C01781=1037.136,384.504,-134.094,173.331,45.031,158.902
C01782=1037.127,384.258,-134.052,173.323,45.027,158.900
C01783=1037.118,384.011,-134.010,173.315,45.023,158.898
C01784=1037.109,383.766,-133.968,173.307,45.019,158.896
C01785=1037.100,383.519,-133.926,173.300,45.015,158.895
C01786=1037.091,383.273,-133.884,173.291,45.011,158.893
C01787=1037.082,383.027,-133.842,173.284,45.007,158.891
C01788=1037.075,382.781,-133.800,173.277,45.004,158.889
C01789=1037.066,382.534,-133.759,173.268,45.000,158.888
C01790=1037.057,382.288,-133.717,173.261,44.996,158.886
C01791=1037.048,382.042,-133.675,173.253,44.991,158.884
C01792=1037.039,381.795,-133.634,173.245,44.988,158.882
C01793=1037.031,381.549,-133.593,173.238,44.984,158.881
C01794=1037.022,381.303,-133.551,173.230,44.980,158.879
C01795=1037.014,381.056,-133.509,173.222,44.976,158.877
C01796=1037.006,380.810,-133.468,173.215,44.972,158.875
C01797=1036.997,380.564,-133.426,173.208,44.968,158.874
C01798=1036.988,380.317,-133.385,173.199,44.965,158.872
C01799=1036.979,380.070,-133.343,173.192,44.961,158.870
C01800=1036.971,379.825,-133.302,173.185,44.957,158.869
C01801=1036.962,379.578,-133.261,173.177,44.953,158.867
C01802=1036.954,379.332,-133.219,173.169,44.950,158.865
C01803=1036.946,379.085,-133.177,173.162,44.946,158.863
C01804=1036.937,378.839,-133.136,173.155,44.942,158.862
C01805=1036.923,378.436,-133.069,173.142,44.936,158.859
C01806=1036.909,378.034,-133.001,173.131,44.930,158.856
C01807=1036.895,377.630,-132.935,173.118,44.924,158.854
C01808=1036.881,377.228,-132.867,173.107,44.918,158.851
C01809=1036.872,376.982,-132.827,173.099,44.915,158.849
C01810=1036.864,376.735,-132.786,173.091,44.911,158.848
C01811=1036.855,376.488,-132.745,173.084,44.907,158.846
C01812=1036.847,376.242,-132.705,173.077,44.904,158.844
C01813=1036.838,375.996,-132.663,173.070,44.900,158.843
C01814=1036.829,375.750,-132.623,173.063,44.896,158.841
C01815=1036.821,375.503,-132.582,173.055,44.893,158.839
C01816=1036.813,375.256,-132.541,173.047,44.889,158.838
C01817=1036.805,375.010,-132.501,173.040,44.886,158.836
C01818=1036.796,374.763,-132.460,173.033,44.883,158.835
C01819=1036.787,374.517,-132.420,173.026,44.879,158.833
C01820=1036.779,374.270,-132.379,173.019,44.876,158.832
C01821=1036.771,374.024,-132.338,173.012,44.872,158.830
C01822=1036.763,373.778,-132.297,173.005,44.869,158.828
C01823=1036.753,373.531,-132.257,172.998,44.865,158.827
C01824=1036.746,373.284,-132.217,172.991,44.862,158.825
C01825=1036.738,373.038,-132.176,172.984,44.858,158.824
C01826=1036.729,372.791,-132.135,172.976,44.855,158.822
C01827=1036.721,372.545,-132.095,172.969,44.851,158.821
C01828=1036.712,372.298,-132.056,172.962,44.848,158.819
C01829=1036.704,372.052,-132.015,172.955,44.845,158.818
C01830=1036.696,371.805,-131.974,172.948,44.841,158.816
C01831=1036.688,371.558,-131.933,172.941,44.838,158.815
C01832=1036.679,371.312,-131.894,172.934,44.835,158.813
C01833=1036.671,371.066,-131.853,172.927,44.832,158.812
C01834=1036.664,370.819,-131.813,172.921,44.828,158.810
C01835=1036.655,370.572,-131.772,172.914,44.825,158.809
C01836=1036.647,370.325,-131.733,172.907,44.821,158.807
C01837=1036.639,370.079,-131.692,172.900,44.818,158.806
C01838=1036.631,369.832,-131.652,172.893,44.814,158.804
C01839=1036.622,369.586,-131.612,172.886,44.811,158.803
C01840=1036.614,369.339,-131.573,172.879,44.808,158.801
C01841=1036.605,369.092,-131.533,172.872,44.805,158.800
C01842=1036.596,368.846,-131.493,172.865,44.802,158.798
C01843=1036.589,368.599,-131.453,172.859,44.799,158.797
C01844=1036.580,368.352,-131.414,172.852,44.796,158.795
C01845=1036.573,368.105,-131.374,172.845,44.792,158.794
C01846=1036.564,367.859,-131.334,172.838,44.789,158.792
C01847=1036.556,367.612,-131.294,172.831,44.786,158.791
C01848=1036.548,367.366,-131.254,172.825,44.783,158.790
C01849=1036.539,367.119,-131.215,172.818,44.780,158.788
C01850=1036.531,366.872,-131.175,172.811,44.777,158.787
C01851=1036.523,366.626,-131.136,172.805,44.774,158.785
C01852=1036.515,366.379,-131.096,172.798,44.771,158.784
C01853=1036.507,366.132,-131.057,172.791,44.768,158.782
C01854=1036.499,365.885,-131.017,172.785,44.764,158.781
C01855=1036.491,365.639,-130.977,172.778,44.761,158.780
C01856=1036.482,365.392,-130.938,172.771,44.758,158.778
C01857=1036.474,365.145,-130.898,172.765,44.755,158.777
C01858=1036.466,364.899,-130.859,172.758,44.752,158.775
C01859=1036.459,364.651,-130.820,172.752,44.749,158.774
C01860=1036.450,364.404,-130.780,172.745,44.746,158.773
C01861=1036.438,364.022,-130.719,172.734,44.741,158.770
C01862=1036.426,363.640,-130.658,172.725,44.737,158.768
C01863=1036.413,363.258,-130.598,172.715,44.732,158.766
C01864=1036.401,362.876,-130.537,172.704,44.728,158.764
C01865=1036.393,362.629,-130.497,172.698,44.724,158.763
C01866=1036.385,362.382,-130.458,172.692,44.721,158.761
C01867=1036.377,362.136,-130.419,172.685,44.719,158.760
C01868=1036.369,361.889,-130.379,172.679,44.716,158.759
C01869=1036.361,361.642,-130.341,172.672,44.712,158.757
C01870=1036.353,361.395,-130.301,172.666,44.710,158.756
C01871=1036.345,361.148,-130.263,172.659,44.707,158.755
C01872=1036.338,360.901,-130.224,172.653,44.704,158.754
C01873=1036.329,360.654,-130.185,172.647,44.701,158.752
C01874=1036.321,360.407,-130.146,172.640,44.699,158.751
C01875=1036.313,360.161,-130.107,172.634,44.695,158.750
C01876=1036.305,359.914,-130.069,172.628,44.693,158.748
C01877=1036.297,359.667,-130.030,172.621,44.691,158.747
C01878=1036.289,359.420,-129.992,172.615,44.687,158.746
C01879=1036.281,359.174,-129.952,172.609,44.685,158.745
C01880=1036.274,358.926,-129.913,172.603,44.681,158.743
C01881=1036.266,358.680,-129.875,172.596,44.679,158.742
C01882=1036.258,358.432,-129.836,172.590,44.676,158.741
C01883=1036.250,358.185,-129.798,172.584,44.674,158.740
C01884=1036.242,357.939,-129.759,172.577,44.671,158.738
C01885=1036.234,357.691,-129.721,172.571,44.668,158.737
C01886=1036.226,357.446,-129.682,172.565,44.666,158.736
C01887=1036.218,357.198,-129.643,172.559,44.663,158.734
C01888=1036.210,356.952,-129.605,172.553,44.660,158.733
C01889=1036.202,356.705,-129.566,172.546,44.657,158.732
C01890=1036.195,356.458,-129.528,172.541,44.655,158.731
C01891=1036.187,356.211,-129.490,172.534,44.652,158.729
C01892=1036.179,355.964,-129.452,172.529,44.649,158.728
C01893=1036.171,355.717,-129.413,172.522,44.647,158.727
C01894=1036.163,355.469,-129.375,172.516,44.644,158.726
C01895=1036.155,355.223,-129.337,172.510,44.642,158.725
C01896=1036.147,354.976,-129.298,172.504,44.639,158.723
C01897=1036.140,354.728,-129.260,172.498,44.636,158.722
C01898=1036.132,354.482,-129.223,172.491,44.634,158.721
C01899=1036.124,354.235,-129.184,172.486,44.631,158.720
C01900=1036.116,353.989,-129.146,172.479,44.629,158.719
C01901=1036.108,353.741,-129.108,172.474,44.626,158.717
C01902=1036.101,353.494,-129.070,172.467,44.624,158.716
C01903=1036.093,353.246,-129.032,172.462,44.621,158.715
C01904=1036.085,353.000,-128.994,172.455,44.618,158.714
C01905=1036.077,352.754,-128.956,172.450,44.616,158.713
C01906=1036.069,352.506,-128.918,172.443,44.614,158.711
C01907=1036.062,352.259,-128.880,172.438,44.611,158.710
C01908=1036.054,352.012,-128.842,172.432,44.608,158.709
C01909=1036.046,351.765,-128.804,172.426,44.606,158.708
C01910=1036.039,351.518,-128.766,172.420,44.604,158.707
C01911=1036.031,351.271,-128.728,172.414,44.601,158.706
C01912=1036.023,351.024,-128.691,172.408,44.598,158.704
C01913=1036.015,350.777,-128.652,172.402,44.596,158.703
C01914=1036.008,350.530,-128.615,172.396,44.594,158.702
C01915=1036.001,350.283,-128.577,172.391,44.591,158.701
C01916=1035.993,350.036,-128.539,172.385,44.589,158.700
C01917=1035.981,349.660,-128.482,172.376,44.585,158.698
C01918=1035.969,349.284,-128.425,172.367,44.581,158.696
C01919=1035.957,348.907,-128.368,172.358,44.578,158.695
C01920=1035.946,348.531,-128.311,172.350,44.574,158.693
C01921=1035.938,348.284,-128.273,172.343,44.572,158.692
C01922=1035.931,348.037,-128.235,172.338,44.570,158.691
C01923=1035.923,347.790,-128.198,172.333,44.567,158.690
C01924=1035.916,347.543,-128.161,172.326,44.565,158.689
C01925=1035.908,347.296,-128.124,172.321,44.563,158.688
C01926=1035.900,347.048,-128.086,172.315,44.560,158.686
C01927=1035.893,346.801,-128.048,172.309,44.558,158.685
C01928=1035.885,346.554,-128.011,172.304,44.556,158.684
C01929=1035.877,346.307,-127.974,172.298,44.553,158.683
C01930=1035.869,346.060,-127.937,172.292,44.551,158.682
C01931=1035.862,345.813,-127.899,172.287,44.549,158.681
C01932=1035.854,345.566,-127.863,172.281,44.547,158.680
C01933=1035.847,345.319,-127.826,172.275,44.545,158.679
C01934=1035.840,345.072,-127.788,172.270,44.542,158.678
C01935=1035.832,344.825,-127.751,172.264,44.540,158.677
C01936=1035.825,344.578,-127.714,172.259,44.538,158.676
C01937=1035.817,344.330,-127.677,172.253,44.536,158.675
C01938=1035.810,344.083,-127.640,172.247,44.533,158.674
C01939=1035.802,343.836,-127.603,172.242,44.531,158.673
C01940=1035.795,343.589,-127.566,172.237,44.529,158.672
C01941=1035.787,343.342,-127.529,172.230,44.527,158.671
C01942=1035.780,343.094,-127.492,172.225,44.525,158.670
C01943=1035.772,342.848,-127.455,172.220,44.522,158.668
C01944=1035.764,342.600,-127.419,172.214,44.520,158.667
C01945=1035.757,342.353,-127.381,172.208,44.518,158.666
C01946=1035.749,342.106,-127.345,172.203,44.516,158.665
C01947=1035.742,341.858,-127.307,172.197,44.514,158.664
C01948=1035.734,341.611,-127.271,172.192,44.512,158.663
C01949=1035.727,341.364,-127.234,172.187,44.510,158.662
C01950=1035.719,341.116,-127.197,172.181,44.508,158.661
C01951=1035.712,340.870,-127.161,172.175,44.506,158.660
C01952=1035.705,340.623,-127.124,172.170,44.503,158.659
C01953=1035.697,340.376,-127.087,172.165,44.502,158.658
C01954=1035.689,340.128,-127.051,172.160,44.500,158.657
C01955=1035.682,339.881,-127.015,172.153,44.498,158.656
C01956=1035.674,339.634,-126.977,172.148,44.496,158.655
C01957=1035.667,339.386,-126.941,172.143,44.493,158.654
C01958=1035.660,339.140,-126.905,172.138,44.492,158.653
C01959=1035.652,338.892,-126.869,172.133,44.490,158.652
C01960=1035.644,338.645,-126.832,172.127,44.488,158.651
C01961=1035.637,338.397,-126.795,172.121,44.486,158.650
C01962=1035.629,338.150,-126.759,172.116,44.483,158.649
C01963=1035.622,337.903,-126.723,172.111,44.482,158.649
C01964=1035.615,337.656,-126.687,172.106,44.480,158.647
C01965=1035.608,337.408,-126.650,172.100,44.477,158.646
C01966=1035.600,337.161,-126.614,172.095,44.476,158.646
C01967=1035.593,336.915,-126.577,172.090,44.474,158.645
C01968=1035.585,336.667,-126.541,172.085,44.472,158.644
C01969=1035.577,336.420,-126.505,172.080,44.470,158.643
C01970=1035.570,336.172,-126.468,172.073,44.468,158.642
C01971=1035.563,335.925,-126.432,172.068,44.466,158.641
C01972=1035.556,335.678,-126.396,172.063,44.464,158.640
C01973=1035.545,335.298,-126.340,172.055,44.461,158.638
C01974=1035.533,334.919,-126.285,172.048,44.458,158.637
C01975=1035.522,334.538,-126.230,172.040,44.455,158.636
C01976=1035.511,334.159,-126.175,172.031,44.453,158.634
C01977=1035.503,333.911,-126.138,172.026,44.451,158.633
C01978=1035.496,333.665,-126.103,172.021,44.449,158.632
C01979=1035.489,333.417,-126.067,172.016,44.447,158.631
C01980=1035.481,333.170,-126.031,172.010,44.445,158.630
C01981=1035.474,332.922,-125.995,172.005,44.444,158.630
C01982=1035.466,332.675,-125.959,172.000,44.442,158.629
C01983=1035.459,332.428,-125.924,171.995,44.440,158.628
C01984=1035.451,332.180,-125.888,171.990,44.438,158.627
C01985=1035.444,331.934,-125.852,171.985,44.437,158.626
C01986=1035.437,331.686,-125.817,171.980,44.435,158.625
C01987=1035.429,331.439,-125.781,171.975,44.433,158.624
C01988=1035.422,331.191,-125.745,171.970,44.431,158.623
C01989=1035.415,330.944,-125.710,171.964,44.429,158.622
C01990=1035.408,330.696,-125.674,171.959,44.428,158.622
C01991=1035.401,330.449,-125.638,171.954,44.426,158.621
C01992=1035.393,330.202,-125.602,171.949,44.424,158.620
C01993=1035.386,329.955,-125.567,171.944,44.423,158.619
C01994=1035.379,329.706,-125.531,171.939,44.421,158.618
C01995=1035.372,329.460,-125.495,171.934,44.419,158.617
C01996=1035.364,329.212,-125.460,171.929,44.418,158.616
C01997=1035.357,328.965,-125.424,171.924,44.416,158.616
C01998=1035.350,328.718,-125.389,171.919,44.414,158.615
C01999=1035.342,328.470,-125.353,171.914,44.412,158.614
C02000=1035.335,328.223,-125.318,171.909,44.411,158.613
C02001=1035.328,327.975,-125.283,171.904,44.409,158.612
C02002=1035.320,327.728,-125.248,171.899,44.407,158.611
C02003=1035.313,327.480,-125.213,171.894,44.406,158.610
C02004=1035.305,327.233,-125.177,171.890,44.404,158.610
C02005=1035.298,326.986,-125.142,171.885,44.403,158.609
C02006=1035.290,326.738,-125.107,171.880,44.401,158.608
C02007=1035.284,326.491,-125.072,171.875,44.400,158.607
C02008=1035.275,326.243,-125.037,171.870,44.398,158.606
C02009=1035.269,325.996,-125.002,171.865,44.397,158.606
C02010=1035.261,325.749,-124.968,171.860,44.395,158.605
C02011=1035.254,325.501,-124.932,171.855,44.394,158.604
C02012=1035.246,325.254,-124.898,171.850,44.392,158.603
C02013=1035.240,325.006,-124.862,171.845,44.390,158.602
C02014=1035.231,324.758,-124.828,171.840,44.389,158.602
C02015=1035.225,324.511,-124.792,171.835,44.388,158.601
C02016=1035.217,324.264,-124.758,171.830,44.386,158.600
C02017=1035.210,324.016,-124.722,171.826,44.384,158.599
C02018=1035.202,323.769,-124.688,171.821,44.383,158.598
C02019=1035.196,323.522,-124.653,171.816,44.382,158.598
C02020=1035.188,323.275,-124.618,171.811,44.380,158.597
C02021=1035.181,323.026,-124.583,171.806,44.379,158.596
C02022=1035.173,322.779,-124.548,171.801,44.377,158.595
C02023=1035.167,322.531,-124.514,171.796,44.376,158.594
C02024=1035.159,322.284,-124.479,171.791,44.374,158.594
C02025=1035.152,322.036,-124.444,171.787,44.373,158.593
C02026=1035.144,321.789,-124.409,171.783,44.372,158.592
C02027=1035.138,321.542,-124.374,171.778,44.370,158.591
C02028=1035.130,321.294,-124.340,171.773,44.368,158.590
C02029=1035.119,320.910,-124.286,171.765,44.366,158.589
C02030=1035.108,320.526,-124.232,171.758,44.364,158.588
C02031=1035.096,320.142,-124.178,171.750,44.362,158.587
C02032=1035.085,319.757,-124.125,171.743,44.360,158.586
C02033=1035.079,319.510,-124.090,171.739,44.358,158.585
C02034=1035.071,319.262,-124.056,171.734,44.357,158.584
C02035=1035.065,319.015,-124.021,171.729,44.356,158.584
C02036=1035.057,318.767,-123.987,171.724,44.354,158.583
C02037=1035.051,318.519,-123.952,171.720,44.353,158.582
C02038=1035.043,318.272,-123.918,171.715,44.351,158.581
C02039=1035.037,318.024,-123.883,171.711,44.350,158.581
C02040=1035.029,317.777,-123.849,171.706,44.349,158.580
C02041=1035.022,317.530,-123.814,171.701,44.347,158.579
C02042=1035.015,317.282,-123.780,171.697,44.346,158.578
C02043=1035.008,317.035,-123.746,171.692,44.344,158.577
C02044=1035.001,316.787,-123.711,171.687,44.343,158.577
C02045=1034.994,316.540,-123.677,171.683,44.342,158.576
C02046=1034.987,316.292,-123.642,171.678,44.340,158.575
C02047=1034.980,316.045,-123.608,171.673,44.339,158.575
C02048=1034.973,315.798,-123.573,171.668,44.338,158.574
C02049=1034.966,315.550,-123.539,171.665,44.337,158.573
C02050=1034.959,315.302,-123.505,171.660,44.335,158.572
C02051=1034.952,315.055,-123.470,171.655,44.334,158.572
C02052=1034.945,314.808,-123.437,171.651,44.332,158.571
C02053=1034.939,314.560,-123.402,171.646,44.331,158.570
C02054=1034.932,314.313,-123.368,171.641,44.330,158.570
C02055=1034.924,314.065,-123.334,171.637,44.328,158.569
C02056=1034.918,313.817,-123.299,171.633,44.327,158.568
C02057=1034.911,313.569,-123.266,171.628,44.326,158.567
C02058=1034.904,313.322,-123.230,171.624,44.325,158.567
C02059=1034.897,313.075,-123.197,171.619,44.324,158.566
C02060=1034.890,312.827,-123.163,171.614,44.322,158.565
C02061=1034.884,312.579,-123.129,171.610,44.321,158.565
C02062=1034.876,312.331,-123.095,171.606,44.320,158.564
C02063=1034.870,312.084,-123.060,171.601,44.318,158.563
C02064=1034.863,311.837,-123.026,171.597,44.317,158.562
C02065=1034.856,311.589,-122.992,171.592,44.316,158.562
C02066=1034.849,311.342,-122.959,171.587,44.315,158.561
C02067=1034.841,311.094,-122.925,171.584,44.314,158.560
C02068=1034.834,310.846,-122.891,171.579,44.313,158.560
C02069=1034.828,310.599,-122.858,171.574,44.312,158.559
C02070=1034.820,310.352,-122.825,171.570,44.310,158.558
C02071=1034.813,310.104,-122.791,171.565,44.309,158.558
C02072=1034.806,309.856,-122.757,171.561,44.308,158.557
C02073=1034.798,309.608,-122.724,171.557,44.307,158.557
C02074=1034.791,309.361,-122.690,171.552,44.306,158.556
C02075=1034.784,309.114,-122.658,171.547,44.305,158.555
C02076=1034.777,308.866,-122.624,171.544,44.304,158.555
C02077=1034.770,308.618,-122.590,171.539,44.303,158.554
C02078=1034.763,308.371,-122.556,171.534,44.302,158.553
C02079=1034.756,308.123,-122.523,171.530,44.301,158.553
C02080=1034.748,307.876,-122.490,171.526,44.300,158.552
C02081=1034.741,307.628,-122.456,171.521,44.299,158.551
C02082=1034.734,307.380,-122.423,171.517,44.297,158.551
C02083=1034.728,307.133,-122.390,171.512,44.296,158.550
C02084=1034.720,306.885,-122.357,171.508,44.295,158.549
C02085=1034.710,306.505,-122.306,171.502,44.294,158.548
C02086=1034.698,306.126,-122.254,171.494,44.292,158.547
C02087=1034.688,305.746,-122.203,171.488,44.291,158.547
C02088=1034.677,305.367,-122.152,171.481,44.290,158.546
C02089=1034.670,305.120,-122.119,171.477,44.288,158.545
C02090=1034.663,304.872,-122.086,171.473,44.287,158.544
C02091=1034.656,304.624,-122.053,171.469,44.286,158.544
C02092=1034.649,304.377,-122.020,171.464,44.285,158.543
C02093=1034.642,304.129,-121.987,171.460,44.284,158.542
C02094=1034.636,303.881,-121.954,171.456,44.283,158.542
C02095=1034.628,303.634,-121.921,171.451,44.282,158.541
C02096=1034.621,303.386,-121.887,171.447,44.281,158.541
C02097=1034.614,303.139,-121.854,171.443,44.280,158.540
C02098=1034.607,302.890,-121.821,171.439,44.280,158.539
C02099=1034.601,302.643,-121.787,171.434,44.279,158.539
C02100=1034.593,302.395,-121.755,171.431,44.277,158.538
C02101=1034.587,302.148,-121.722,171.426,44.276,158.538
C02102=1034.580,301.900,-121.688,171.422,44.276,158.537
C02103=1034.573,301.653,-121.656,171.418,44.275,158.536
C02104=1034.566,301.405,-121.623,171.414,44.273,158.536
C02105=1034.559,301.158,-121.590,171.409,44.272,158.535
C02106=1034.552,300.909,-121.557,171.406,44.272,158.535
C02107=1034.546,300.662,-121.524,171.401,44.271,158.534
C02108=1034.538,300.414,-121.491,171.397,44.270,158.533
C02109=1034.532,300.167,-121.458,171.393,44.269,158.533
C02110=1034.525,299.919,-121.425,171.389,44.268,158.532
C02111=1034.519,299.671,-121.392,171.384,44.267,158.532
C02112=1034.511,299.423,-121.359,171.380,44.266,158.531
C02113=1034.505,299.175,-121.327,171.376,44.265,158.530
C02114=1034.498,298.928,-121.294,171.372,44.264,158.530
C02115=1034.490,298.680,-121.261,171.367,44.264,158.529
C02116=1034.484,298.433,-121.228,171.364,44.262,158.529
C02117=1034.477,298.184,-121.195,171.359,44.261,158.528
C02118=1034.471,297.937,-121.162,171.355,44.261,158.528
C02119=1034.464,297.690,-121.130,171.352,44.260,158.527
C02120=1034.457,297.441,-121.097,171.347,44.259,158.526
C02121=1034.451,297.194,-121.064,171.343,44.258,158.526
C02122=1034.444,296.946,-121.031,171.339,44.257,158.525
C02123=1034.437,296.698,-120.999,171.335,44.256,158.525
C02124=1034.431,296.451,-120.966,171.330,44.255,158.524
C02125=1034.424,296.203,-120.933,171.327,44.255,158.524
C02126=1034.417,295.955,-120.901,171.323,44.253,158.523
C02127=1034.410,295.707,-120.868,171.318,44.252,158.522
C02128=1034.404,295.460,-120.835,171.315,44.252,158.522
C02129=1034.397,295.211,-120.802,171.310,44.251,158.521
C02130=1034.390,294.964,-120.770,171.307,44.250,158.521
C02131=1034.384,294.717,-120.737,171.303,44.249,158.520
C02132=1034.376,294.469,-120.705,171.298,44.248,158.520
C02133=1034.370,294.221,-120.672,171.295,44.248,158.519
C02134=1034.363,293.973,-120.641,171.290,44.247,158.518
C02135=1034.356,293.726,-120.609,171.286,44.246,158.518
C02136=1034.349,293.478,-120.575,171.283,44.246,158.518
C02137=1034.343,293.230,-120.544,171.278,44.245,158.517
C02138=1034.336,292.982,-120.511,171.275,44.244,158.516
C02139=1034.329,292.734,-120.479,171.270,44.243,158.516
C02140=1034.322,292.487,-120.447,171.266,44.242,158.515
C02141=1034.312,292.124,-120.400,171.261,44.241,158.515
C02142=1034.301,291.761,-120.353,171.255,44.241,158.514
C02143=1034.292,291.399,-120.306,171.249,44.239,158.513
C02144=1034.282,291.036,-120.259,171.243,44.238,158.512
C02145=1034.275,290.789,-120.227,171.240,44.238,158.512
C02146=1034.268,290.540,-120.195,171.235,44.237,158.511
C02147=1034.261,290.293,-120.163,171.231,44.236,158.511
C02148=1034.254,290.045,-120.130,171.228,44.235,158.510
C02149=1034.248,289.797,-120.098,171.223,44.235,158.510
C02150=1034.241,289.549,-120.067,171.220,44.234,158.509
C02151=1034.234,289.301,-120.034,171.216,44.233,158.509
C02152=1034.227,289.053,-120.003,171.212,44.233,158.508
C02153=1034.220,288.806,-119.971,171.208,44.232,158.508
C02154=1034.214,288.558,-119.939,171.205,44.231,158.507
C02155=1034.207,288.311,-119.907,171.200,44.231,158.507
C02156=1034.200,288.063,-119.875,171.196,44.230,158.506
C02157=1034.193,287.814,-119.843,171.193,44.229,158.506
C02158=1034.186,287.567,-119.811,171.188,44.229,158.505
C02159=1034.180,287.319,-119.779,171.185,44.228,158.505
C02160=1034.173,287.071,-119.748,171.181,44.228,158.504
C02161=1034.166,286.823,-119.716,171.177,44.227,158.504
C02162=1034.159,286.576,-119.684,171.173,44.226,158.503
C02163=1034.153,286.328,-119.653,171.170,44.226,158.503
C02164=1034.145,286.079,-119.621,171.165,44.225,158.502
C02165=1034.138,285.832,-119.589,171.162,44.225,158.502
C02166=1034.132,285.584,-119.557,171.158,44.224,158.501
C02167=1034.125,285.336,-119.526,171.154,44.224,158.501
C02168=1034.118,285.088,-119.495,171.150,44.223,158.500
C02169=1034.111,284.840,-119.463,171.147,44.223,158.500
C02170=1034.105,284.592,-119.432,171.142,44.222,158.500
C02171=1034.098,284.344,-119.400,171.139,44.221,158.499
C02172=1034.091,284.096,-119.369,171.135,44.221,158.499
C02173=1034.084,283.848,-119.337,171.131,44.220,158.498
C02174=1034.077,283.601,-119.305,171.127,44.220,158.498
C02175=1034.070,283.353,-119.274,171.123,44.219,158.497
C02176=1034.063,283.105,-119.242,171.120,44.219,158.497
C02177=1034.057,282.857,-119.211,171.115,44.218,158.496
C02178=1034.049,282.609,-119.180,171.112,44.217,158.496
C02179=1034.043,282.361,-119.148,171.108,44.217,158.495
C02180=1034.036,282.113,-119.117,171.104,44.216,158.495
C02181=1034.029,281.866,-119.086,171.100,44.216,158.494
C02182=1034.022,281.618,-119.054,171.097,44.215,158.494
C02183=1034.016,281.369,-119.023,171.093,44.215,158.493
C02184=1034.009,281.121,-118.992,171.089,44.215,158.493
C02185=1034.002,280.873,-118.961,171.086,44.214,158.493
C02186=1033.996,280.625,-118.929,171.082,44.213,158.492
C02187=1033.989,280.378,-118.898,171.079,44.213,158.492
C02188=1033.982,280.130,-118.866,171.075,44.212,158.491
C02189=1033.976,279.882,-118.835,171.071,44.212,158.491
C02190=1033.969,279.634,-118.803,171.067,44.211,158.490
C02191=1033.962,279.386,-118.772,171.064,44.211,158.490
C02192=1033.956,279.138,-118.742,171.060,44.211,158.490
C02193=1033.950,278.890,-118.710,171.056,44.210,158.489
C02194=1033.943,278.642,-118.679,171.052,44.209,158.489
C02195=1033.935,278.395,-118.648,171.049,44.209,158.488
C02196=1033.929,278.147,-118.616,171.045,44.208,158.488
C02197=1033.920,277.796,-118.573,171.040,44.208,158.487
C02198=1033.910,277.445,-118.529,171.035,44.207,158.486
C02199=1033.900,277.095,-118.485,171.029,44.207,158.486
C02200=1033.891,276.744,-118.441,171.025,44.206,158.485
C02201=1033.883,276.497,-118.410,171.020,44.206,158.485
C02202=1033.877,276.248,-118.380,171.017,44.205,158.484
C02203=1033.870,276.000,-118.348,171.013,44.205,158.484
C02204=1033.864,275.752,-118.318,171.010,44.205,158.484
C02205=1033.856,275.504,-118.287,171.007,44.204,158.483
C02206=1033.850,275.256,-118.256,171.002,44.204,158.483
C02207=1033.844,275.009,-118.225,170.999,44.204,158.482
C02208=1033.836,274.761,-118.194,170.995,44.203,158.482
C02209=1033.830,274.513,-118.163,170.992,44.202,158.482
C02210=1033.823,274.265,-118.132,170.988,44.202,158.481
C02211=1033.816,274.016,-118.102,170.985,44.202,158.481
C02212=1033.809,273.768,-118.070,170.980,44.201,158.480
C02213=1033.804,273.521,-118.040,170.977,44.201,158.480
C02214=1033.796,273.272,-118.010,170.974,44.201,158.480
C02215=1033.790,273.025,-117.979,170.970,44.200,158.479
C02216=1033.782,272.776,-117.948,170.967,44.200,158.479
C02217=1033.776,272.528,-117.917,170.963,44.199,158.478
C02218=1033.770,272.281,-117.887,170.959,44.199,158.478
C02219=1033.763,272.032,-117.856,170.956,44.199,158.478
C02220=1033.756,271.784,-117.825,170.952,44.199,158.477
C02221=1033.749,271.536,-117.795,170.949,44.198,158.477
C02222=1033.742,271.288,-117.764,170.945,44.198,158.476
C02223=1033.736,271.041,-117.734,170.942,44.197,158.476
C02224=1033.729,270.792,-117.703,170.939,44.197,158.476
C02225=1033.722,270.544,-117.673,170.934,44.197,158.475
C02226=1033.716,270.296,-117.642,170.931,44.196,158.475
C02227=1033.709,270.049,-117.612,170.927,44.196,158.474
C02228=1033.702,269.800,-117.581,170.924,44.196,158.474
C02229=1033.695,269.552,-117.551,170.921,44.196,158.474
C02230=1033.689,269.303,-117.520,170.917,44.195,158.473
C02231=1033.682,269.056,-117.490,170.914,44.195,158.473
C02232=1033.675,268.808,-117.459,170.910,44.194,158.472
C02233=1033.668,268.560,-117.429,170.906,44.195,158.472
C02234=1033.662,268.312,-117.399,170.903,44.194,158.472
C02235=1033.655,268.064,-117.368,170.899,44.194,158.471
C02236=1033.648,267.816,-117.338,170.896,44.194,158.471
C02237=1033.642,267.567,-117.308,170.893,44.193,158.471
C02238=1033.635,267.320,-117.278,170.889,44.193,158.470
C02239=1033.628,267.071,-117.248,170.886,44.193,158.470
C02240=1033.622,266.823,-117.217,170.883,44.193,158.470
C02241=1033.615,266.575,-117.187,170.879,44.192,158.469
C02242=1033.608,266.327,-117.157,170.876,44.192,158.469
C02243=1033.602,266.079,-117.126,170.871,44.192,158.468
C02244=1033.595,265.831,-117.097,170.868,44.192,158.468
C02245=1033.588,265.583,-117.066,170.865,44.192,158.468
C02246=1033.581,265.335,-117.036,170.861,44.192,158.467
C02247=1033.575,265.087,-117.006,170.858,44.191,158.467
C02248=1033.568,264.839,-116.976,170.855,44.191,158.467
C02249=1033.561,264.591,-116.946,170.851,44.191,158.466
C02250=1033.555,264.343,-116.915,170.848,44.190,158.466
C02251=1033.548,264.094,-116.885,170.845,44.190,158.466
C02252=1033.541,263.847,-116.856,170.841,44.190,158.465
C02253=1033.532,263.501,-116.814,170.836,44.190,158.465
C02254=1033.522,263.155,-116.773,170.831,44.190,158.464
C02255=1033.513,262.808,-116.730,170.827,44.189,158.464
C02256=1033.504,262.463,-116.688,170.822,44.189,158.463
C02257=1033.497,262.215,-116.659,170.819,44.189,158.463
C02258=1033.490,261.966,-116.629,170.816,44.189,158.463
C02259=1033.484,261.719,-116.598,170.812,44.189,158.462
C02260=1033.477,261.470,-116.568,170.809,44.188,158.462
C02261=1033.471,261.222,-116.539,170.806,44.188,158.462
C02262=1033.464,260.974,-116.509,170.801,44.188,158.461
C02263=1033.457,260.726,-116.479,170.798,44.188,158.461
C02264=1033.450,260.478,-116.451,170.795,44.188,158.461
C02265=1033.442,260.230,-116.420,170.792,44.188,158.460
C02266=1033.436,259.982,-116.391,170.788,44.188,158.460
C02267=1033.429,259.734,-116.361,170.785,44.187,158.460
C02268=1033.422,259.486,-116.331,170.781,44.187,158.459
C02269=1033.416,259.237,-116.302,170.778,44.187,158.459
C02270=1033.408,258.989,-116.272,170.775,44.187,158.459
C02271=1033.401,258.741,-116.243,170.772,44.187,158.458
C02272=1033.394,258.493,-116.213,170.768,44.187,158.458
C02273=1033.388,258.245,-116.184,170.765,44.187,158.458
C02274=1033.381,257.997,-116.154,170.762,44.187,158.458
C02275=1033.375,257.748,-116.125,170.759,44.187,158.457
C02276=1033.368,257.500,-116.096,170.755,44.187,158.457
C02277=1033.361,257.252,-116.066,170.752,44.187,158.457
C02278=1033.354,257.004,-116.037,170.749,44.187,158.456
C02279=1033.347,256.756,-116.007,170.745,44.187,158.456
C02280=1033.340,256.507,-115.978,170.742,44.187,158.456
C02281=1033.334,256.260,-115.948,170.739,44.187,158.455
C02282=1033.327,256.011,-115.919,170.735,44.187,158.455
C02283=1033.321,255.763,-115.890,170.732,44.187,158.455
C02284=1033.313,255.515,-115.860,170.729,44.186,158.454
C02285=1033.306,255.267,-115.831,170.726,44.186,158.454
C02286=1033.300,255.018,-115.802,170.722,44.186,158.454
C02287=1033.293,254.770,-115.772,170.719,44.186,158.453
C02288=1033.286,254.522,-115.743,170.716,44.186,158.453
C02289=1033.280,254.273,-115.714,170.713,44.186,158.453
C02290=1033.273,254.026,-115.684,170.709,44.186,158.453
C02291=1033.266,253.777,-115.655,170.706,44.186,158.452
C02292=1033.260,253.529,-115.626,170.703,44.186,158.452
C02293=1033.253,253.280,-115.597,170.699,44.186,158.452
C02294=1033.246,253.033,-115.567,170.696,44.186,158.451
C02295=1033.240,252.785,-115.538,170.693,44.186,158.451
C02296=1033.233,252.536,-115.508,170.690,44.186,158.451
C02297=1033.226,252.288,-115.480,170.686,44.186,158.450
C02298=1033.219,252.040,-115.450,170.683,44.186,158.450
C02299=1033.213,251.792,-115.421,170.680,44.186,158.450
C02300=1033.206,251.544,-115.392,170.677,44.186,158.450
C02301=1033.200,251.295,-115.362,170.673,44.186,158.449
C02302=1033.193,251.047,-115.333,170.670,44.186,158.449
C02303=1033.186,250.799,-115.305,170.668,44.186,158.449
C02304=1033.179,250.551,-115.275,170.664,44.186,158.448
C02305=1033.173,250.303,-115.246,170.661,44.186,158.448
C02306=1033.167,250.054,-115.217,170.658,44.186,158.448
C02307=1033.160,249.806,-115.187,170.655,44.186,158.448
C02308=1033.153,249.558,-115.159,170.651,44.186,158.447
C02309=1033.144,249.210,-115.117,170.647,44.186,158.447
C02310=1033.135,248.863,-115.077,170.643,44.186,158.447
C02311=1033.126,248.515,-115.036,170.638,44.186,158.446
C02312=1033.117,248.169,-114.996,170.634,44.186,158.446
C02313=1033.109,247.920,-114.967,170.631,44.186,158.445
C02314=1033.103,247.672,-114.938,170.627,44.186,158.445
C02315=1033.097,247.424,-114.909,170.624,44.186,158.445
C02316=1033.091,247.176,-114.880,170.621,44.186,158.445
C02317=1033.084,246.927,-114.851,170.618,44.186,158.444
C02318=1033.077,246.679,-114.822,170.616,44.186,158.444
C02319=1033.070,246.431,-114.793,170.612,44.186,158.444
C02320=1033.064,246.183,-114.764,170.609,44.186,158.444
C02321=1033.058,245.935,-114.735,170.606,44.186,158.443
C02322=1033.051,245.686,-114.706,170.603,44.186,158.443
C02323=1033.044,245.438,-114.677,170.599,44.186,158.443
C02324=1033.038,245.190,-114.648,170.596,44.186,158.442
C02325=1033.032,244.942,-114.619,170.594,44.186,158.442
C02326=1033.025,244.694,-114.590,170.590,44.186,158.442
C02327=1033.018,244.445,-114.561,170.587,44.186,158.441
C02328=1033.012,244.196,-114.533,170.584,44.186,158.441
C02329=1033.006,243.948,-114.504,170.581,44.186,158.441
C02330=1032.999,243.700,-114.475,170.578,44.186,158.441
C02331=1032.992,243.452,-114.446,170.574,44.186,158.440
C02332=1032.985,243.203,-114.418,170.572,44.186,158.440
C02333=1032.979,242.955,-114.389,170.569,44.187,158.440
C02334=1032.972,242.707,-114.361,170.566,44.187,158.440
C02335=1032.966,242.459,-114.332,170.563,44.187,158.439
C02336=1032.959,242.211,-114.304,170.559,44.187,158.439
C02337=1032.952,241.962,-114.275,170.556,44.187,158.439
C02338=1032.945,241.714,-114.246,170.554,44.187,158.439
C02339=1032.939,241.465,-114.218,170.551,44.187,158.438
C02340=1032.932,241.217,-114.189,170.547,44.187,158.438
C02341=1032.926,240.969,-114.160,170.544,44.187,158.438
C02342=1032.919,240.721,-114.133,170.541,44.188,158.438
C02343=1032.913,240.473,-114.104,170.538,44.188,158.437
C02344=1032.906,240.223,-114.075,170.536,44.187,158.437
C02345=1032.899,239.975,-114.046,170.533,44.188,158.437
C02346=1032.892,239.728,-114.018,170.529,44.188,158.437
C02347=1032.886,239.479,-113.990,170.526,44.188,158.436
C02348=1032.879,239.231,-113.962,170.523,44.188,158.436
C02349=1032.873,238.983,-113.933,170.520,44.188,158.436
C02350=1032.866,238.735,-113.905,170.517,44.188,158.436
C02351=1032.859,238.486,-113.877,170.514,44.189,158.436
C02352=1032.852,238.237,-113.849,170.511,44.189,158.435
C02353=1032.846,237.989,-113.820,170.508,44.189,158.435
C02354=1032.839,237.741,-113.792,170.505,44.189,158.435
C02355=1032.832,237.493,-113.764,170.502,44.189,158.435
C02356=1032.826,237.244,-113.736,170.499,44.190,158.434
C02357=1032.819,236.996,-113.707,170.496,44.190,158.434
C02358=1032.812,236.748,-113.679,170.493,44.190,158.434
C02359=1032.806,236.499,-113.652,170.490,44.190,158.434
C02360=1032.798,236.251,-113.623,170.487,44.190,158.433
C02361=1032.792,236.002,-113.595,170.485,44.191,158.433
C02362=1032.785,235.754,-113.567,170.481,44.191,158.433
C02363=1032.778,235.506,-113.538,170.478,44.191,158.433
C02364=1032.772,235.257,-113.511,170.475,44.191,158.433
C02365=1032.762,234.904,-113.471,170.471,44.191,158.432
C02366=1032.753,234.551,-113.430,170.466,44.192,158.432
C02367=1032.743,234.198,-113.391,170.462,44.192,158.432
C02368=1032.734,233.845,-113.351,170.458,44.193,158.431
C02369=1032.727,233.596,-113.323,170.456,44.192,158.431
C02370=1032.721,233.348,-113.294,170.453,44.193,158.431
C02371=1032.714,233.099,-113.267,170.450,44.193,158.431
C02372=1032.707,232.851,-113.238,170.446,44.193,158.430
C02373=1032.701,232.603,-113.211,170.444,44.193,158.430
C02374=1032.694,232.354,-113.183,170.441,44.193,158.430
C02375=1032.688,232.106,-113.155,170.438,44.194,158.430
C02376=1032.681,231.857,-113.127,170.435,44.194,158.429
C02377=1032.675,231.610,-113.099,170.433,44.194,158.429
C02378=1032.668,231.362,-113.071,170.429,44.194,158.429
C02379=1032.662,231.113,-113.043,170.426,44.195,158.429
C02380=1032.655,230.865,-113.016,170.423,44.195,158.429
C02381=1032.648,230.616,-112.988,170.421,44.195,158.429
C02382=1032.641,230.368,-112.960,170.418,44.195,158.428
C02383=1032.635,230.119,-112.932,170.415,44.196,158.428
C02384=1032.628,229.871,-112.905,170.411,44.196,158.428
C02385=1032.621,229.623,-112.877,170.409,44.196,158.428
C02386=1032.615,229.374,-112.849,170.406,44.196,158.427
C02387=1032.608,229.126,-112.821,170.403,44.197,158.427
C02388=1032.601,228.878,-112.793,170.400,44.197,158.427
C02389=1032.595,228.629,-112.765,170.398,44.197,158.427
C02390=1032.588,228.381,-112.737,170.395,44.197,158.427
C02391=1032.582,228.132,-112.709,170.392,44.198,158.426
C02392=1032.575,227.884,-112.681,170.388,44.198,158.426
C02393=1032.568,227.636,-112.654,170.386,44.198,158.426
C02394=1032.561,227.387,-112.627,170.383,44.199,158.426
C02395=1032.555,227.138,-112.600,170.380,44.199,158.426
C02396=1032.548,226.890,-112.572,170.378,44.199,158.425
C02397=1032.542,226.642,-112.544,170.375,44.200,158.425
C02398=1032.534,226.394,-112.517,170.372,44.200,158.425
C02399=1032.528,226.145,-112.490,170.369,44.200,158.425
C02400=1032.521,225.897,-112.462,170.367,44.201,158.425
C02401=1032.515,225.648,-112.435,170.363,44.201,158.424
C02402=1032.508,225.399,-112.407,170.360,44.201,158.424
C02403=1032.501,225.151,-112.380,170.357,44.202,158.424
C02404=1032.494,224.903,-112.352,170.355,44.202,158.424
C02405=1032.487,224.654,-112.325,170.352,44.202,158.424
C02406=1032.481,224.406,-112.297,170.349,44.203,158.424
C02407=1032.475,224.158,-112.270,170.347,44.203,158.423
C02408=1032.467,223.910,-112.243,170.344,44.203,158.423
C02409=1032.461,223.661,-112.215,170.341,44.204,158.423
C02410=1032.454,223.413,-112.188,170.338,44.204,158.423
C02411=1032.448,223.164,-112.161,170.335,44.204,158.423
C02412=1032.441,222.915,-112.133,170.332,44.205,158.423
C02413=1032.434,222.667,-112.106,170.329,44.205,158.422
C02414=1032.427,222.419,-112.078,170.327,44.205,158.422
C02415=1032.421,222.170,-112.051,170.324,44.206,158.422
C02416=1032.414,221.922,-112.024,170.321,44.206,158.422
C02417=1032.407,221.674,-111.996,170.319,44.206,158.422
C02418=1032.401,221.425,-111.969,170.316,44.207,158.421
C02419=1032.395,221.177,-111.942,170.312,44.207,158.421
C02420=1032.388,220.928,-111.914,170.310,44.207,158.421
C02421=1032.378,220.568,-111.875,170.306,44.208,158.421
C02422=1032.369,220.207,-111.835,170.302,44.208,158.421
C02423=1032.359,219.846,-111.796,170.298,44.209,158.420
C02424=1032.349,219.485,-111.757,170.294,44.209,158.420
C02425=1032.343,219.237,-111.729,170.292,44.210,158.420
C02426=1032.336,218.988,-111.703,170.288,44.210,158.420
C02427=1032.329,218.740,-111.675,170.285,44.211,158.420
C02428=1032.322,218.492,-111.649,170.283,44.211,158.419
C02429=1032.316,218.243,-111.621,170.280,44.211,158.419
C02430=1032.309,217.994,-111.595,170.277,44.212,158.419
C02431=1032.302,217.746,-111.567,170.275,44.212,158.419
C02432=1032.295,217.497,-111.540,170.272,44.213,158.419
C02433=1032.289,217.249,-111.513,170.269,44.213,158.419
C02434=1032.282,217.001,-111.487,170.267,44.213,158.418
C02435=1032.275,216.752,-111.459,170.264,44.214,158.418
C02436=1032.268,216.503,-111.433,170.261,44.214,158.418
C02437=1032.262,216.255,-111.406,170.259,44.215,158.418
C02438=1032.255,216.007,-111.379,170.256,44.215,158.418
C02439=1032.248,215.758,-111.352,170.253,44.215,158.418
C02440=1032.241,215.510,-111.325,170.250,44.216,158.418
C02441=1032.235,215.261,-111.298,170.247,44.216,158.417
C02442=1032.228,215.013,-111.272,170.245,44.217,158.417
C02443=1032.221,214.764,-111.244,170.242,44.217,158.417
C02444=1032.215,214.516,-111.218,170.239,44.218,158.417
C02445=1032.208,214.267,-111.191,170.237,44.218,158.417
C02446=1032.201,214.019,-111.164,170.234,44.218,158.417
C02447=1032.195,213.771,-111.137,170.232,44.219,158.416
C02448=1032.188,213.522,-111.111,170.229,44.219,158.416
C02449=1032.181,213.273,-111.083,170.226,44.220,158.416
C02450=1032.175,213.025,-111.057,170.223,44.220,158.416
C02451=1032.169,212.776,-111.030,170.220,44.220,158.416
C02452=1032.161,212.528,-111.003,170.218,44.221,158.416
C02453=1032.155,212.280,-110.976,170.215,44.221,158.416
C02454=1032.148,212.031,-110.950,170.212,44.222,158.415
C02455=1032.142,211.782,-110.923,170.210,44.222,158.415
C02456=1032.135,211.535,-110.896,170.207,44.223,158.415
C02457=1032.129,211.286,-110.869,170.205,44.223,158.415
C02458=1032.122,211.037,-110.842,170.202,44.223,158.415
C02459=1032.115,210.789,-110.816,170.199,44.224,158.415
C02460=1032.109,210.540,-110.789,170.197,44.224,158.415
C02461=1032.102,210.291,-110.763,170.194,44.225,158.414
C02462=1032.095,210.044,-110.736,170.192,44.225,158.414
C02463=1032.088,209.794,-110.709,170.189,44.226,158.414
C02464=1032.082,209.546,-110.683,170.187,44.226,158.414
C02465=1032.075,209.298,-110.657,170.184,44.227,158.414
C02466=1032.068,209.049,-110.630,170.181,44.228,158.414
C02467=1032.062,208.801,-110.604,170.178,44.227,158.413
C02468=1032.055,208.552,-110.577,170.175,44.228,158.413
C02469=1032.048,208.303,-110.551,170.173,44.228,158.413
C02470=1032.041,208.055,-110.525,170.170,44.229,158.413
C02471=1032.035,207.806,-110.498,170.167,44.230,158.413
C02472=1032.028,207.558,-110.472,170.165,44.230,158.413
C02473=1032.021,207.310,-110.444,170.162,44.231,158.413
C02474=1032.014,207.061,-110.418,170.160,44.231,158.413
C02475=1032.008,206.813,-110.391,170.157,44.232,158.412
C02476=1032.001,206.564,-110.365,170.155,44.232,158.412
C02477=1031.991,206.209,-110.328,170.151,44.233,158.412
C02478=1031.981,205.854,-110.290,170.147,44.234,158.412
C02479=1031.972,205.500,-110.253,170.144,44.234,158.412
C02480=1031.963,205.144,-110.215,170.140,44.235,158.412
C02481=1031.937,204.095,-110.110,169.795,44.131,158.359
C02482=1031.930,203.847,-110.085,169.792,44.133,158.359
C02483=1031.924,203.597,-110.060,169.789,44.134,158.359
C02484=1031.918,203.349,-110.035,169.785,44.135,158.359
C02485=1031.912,203.101,-110.010,169.781,44.136,158.359
C02486=1031.906,202.852,-109.986,169.777,44.137,158.359
C02487=1031.900,202.603,-109.960,169.774,44.139,158.359
C02488=1031.894,202.354,-109.936,169.770,44.140,158.359
C02489=1031.889,202.106,-109.911,169.767,44.142,158.359
C02490=1031.882,201.857,-109.886,169.764,44.143,158.359
C02491=1031.876,201.608,-109.861,169.760,44.144,158.358
C02492=1031.870,201.360,-109.836,169.756,44.145,158.358
C02493=1031.864,201.111,-109.812,169.753,44.146,158.358
C02494=1031.858,200.862,-109.786,169.749,44.148,158.358
C02495=1031.852,200.613,-109.762,169.745,44.149,158.358
C02496=1031.846,200.365,-109.737,169.742,44.151,158.358
C02497=1031.840,200.116,-109.713,169.739,44.152,158.358
C02498=1031.833,199.867,-109.688,169.735,44.153,158.358
C02499=1031.827,199.618,-109.663,169.731,44.155,158.358
C02500=1031.821,199.370,-109.640,169.728,44.156,158.358
C02501=1031.815,199.121,-109.614,169.725,44.157,158.358
C02502=1031.808,198.872,-109.590,169.721,44.159,158.358
C02503=1031.802,198.623,-109.566,169.717,44.160,158.358
C02504=1031.796,198.375,-109.541,169.714,44.162,158.358
C02505=1031.790,198.126,-109.517,169.711,44.164,158.358
C02506=1031.783,197.877,-109.493,169.707,44.165,158.358
C02507=1031.778,197.629,-109.468,169.704,44.166,158.358
C02508=1031.771,197.380,-109.444,169.700,44.168,158.358
C02509=1031.765,197.131,-109.419,169.696,44.169,158.358
C02510=1031.759,196.882,-109.395,169.693,44.170,158.358
C02511=1031.753,196.634,-109.370,169.690,44.172,158.358
C02512=1031.746,196.385,-109.346,169.686,44.173,158.358
C02513=1031.741,196.136,-109.322,169.683,44.175,158.358
C02514=1031.734,195.887,-109.298,169.679,44.177,158.358
C02515=1031.729,195.639,-109.273,169.676,44.178,158.358
C02516=1031.722,195.390,-109.249,169.673,44.179,158.358
C02517=1031.716,195.141,-109.224,169.669,44.181,158.358
C02518=1031.710,194.893,-109.200,169.665,44.182,158.358
C02519=1031.704,194.643,-109.176,169.662,44.183,158.358
C02520=1031.698,194.395,-109.152,169.658,44.185,158.358
C02521=1031.692,194.146,-109.128,169.655,44.187,158.358
C02522=1031.685,193.898,-109.103,169.652,44.188,158.358
C02523=1031.680,193.649,-109.079,169.648,44.190,158.358
C02524=1031.674,193.400,-109.055,169.645,44.191,158.358
C02525=1031.668,193.151,-109.030,169.642,44.192,158.358
C02526=1031.662,192.902,-109.006,169.638,44.194,158.358
C02527=1031.656,192.654,-108.982,169.635,44.195,158.358
C02528=1031.650,192.405,-108.958,169.631,44.197,158.358
C02529=1031.644,192.156,-108.934,169.628,44.199,158.358
C02530=1031.638,191.907,-108.910,169.625,44.200,158.358
C02531=1031.632,191.659,-108.885,169.621,44.201,158.358
C02532=1031.626,191.410,-108.861,169.618,44.203,158.358
C02533=1031.620,191.161,-108.838,169.615,44.205,158.358
C02534=1031.614,190.912,-108.813,169.612,44.206,158.358
C02535=1031.608,190.664,-108.789,169.608,44.207,158.358
C02536=1031.602,190.415,-108.765,169.604,44.209,158.358
C02537=1031.596,190.166,-108.741,169.601,44.210,158.358
C02538=1031.590,189.917,-108.717,169.597,44.211,158.358
C02539=1031.584,189.669,-108.693,169.595,44.213,158.358
C02540=1031.578,189.419,-108.668,169.591,44.215,158.358
C02541=1031.572,189.171,-108.645,169.588,44.216,158.358
C02542=1031.565,188.888,-108.617,169.584,44.218,158.358
C02543=1031.558,188.604,-108.589,169.581,44.220,158.358
C02544=1031.552,188.320,-108.562,169.576,44.221,158.358
C02545=1031.545,188.037,-108.535,169.572,44.223,158.358
C02546=1031.539,187.788,-108.510,169.570,44.225,158.358
C02547=1031.533,187.539,-108.487,169.566,44.226,158.358
C02548=1031.527,187.291,-108.463,169.563,44.227,158.358
C02549=1031.521,187.041,-108.439,169.559,44.229,158.358
C02550=1031.516,186.792,-108.415,169.557,44.231,158.358
C02551=1031.509,186.543,-108.391,169.553,44.232,158.358
C02552=1031.504,186.295,-108.367,169.550,44.233,158.358
C02553=1031.498,186.047,-108.343,169.546,44.235,158.358
C02554=1031.491,185.797,-108.320,169.544,44.237,158.358
C02555=1031.486,185.548,-108.295,169.540,44.238,158.358
C02556=1031.480,185.300,-108.272,169.537,44.239,158.358
C02557=1031.474,185.051,-108.247,169.533,44.241,158.358
C02558=1031.468,184.803,-108.224,169.531,44.243,158.358
C02559=1031.463,184.553,-108.200,169.527,44.244,158.358
C02560=1031.456,184.304,-108.176,169.524,44.245,158.358
C02561=1031.450,184.056,-108.152,169.520,44.247,158.358
C02562=1031.445,183.808,-108.128,169.517,44.249,158.358
C02563=1031.439,183.558,-108.105,169.515,44.250,158.358
C02564=1031.433,183.309,-108.080,169.511,44.251,158.358
C02565=1031.427,183.061,-108.057,169.508,44.253,158.358
C02566=1031.421,182.811,-108.033,169.504,44.255,158.358
C02567=1031.415,182.563,-108.010,169.502,44.256,158.358
C02568=1031.409,182.314,-107.987,169.498,44.258,158.358
C02569=1031.403,182.065,-107.963,169.494,44.260,158.358
C02570=1031.396,181.817,-107.940,169.492,44.262,158.358
C02571=1031.391,181.568,-107.918,169.488,44.264,158.358
C02572=1031.384,181.319,-107.894,169.485,44.265,158.358
C02573=1031.378,181.070,-107.871,169.482,44.267,158.359
C02574=1031.372,180.821,-107.847,169.479,44.268,158.359
C02575=1031.366,180.572,-107.824,169.475,44.270,158.359
C02576=1031.359,180.324,-107.801,169.473,44.272,158.359
C02577=1031.353,180.075,-107.777,169.469,44.274,158.359
C02578=1031.347,179.826,-107.754,169.466,44.276,158.359
C02579=1031.341,179.577,-107.731,169.462,44.277,158.359
C02580=1031.335,179.328,-107.707,169.460,44.279,158.359
C02581=1031.329,179.079,-107.684,169.456,44.281,158.359
C02582=1031.322,178.831,-107.661,169.452,44.283,158.359
C02583=1031.316,178.582,-107.638,169.450,44.284,158.359
C02584=1031.310,178.332,-107.615,169.446,44.286,158.359
C02585=1031.304,178.084,-107.591,169.443,44.288,158.359
C02586=1031.298,177.835,-107.568,169.440,44.290,158.359
C02587=1031.291,177.586,-107.546,169.437,44.291,158.359
C02588=1031.285,177.338,-107.522,169.435,44.293,158.360
C02589=1031.279,177.089,-107.499,169.431,44.294,158.359
C02590=1031.274,176.840,-107.476,169.428,44.296,158.360
C02591=1031.267,176.590,-107.453,169.425,44.298,158.360
C02592=1031.261,176.342,-107.430,169.422,44.300,158.360
C02593=1031.255,176.093,-107.407,169.418,44.302,158.360
C02594=1031.249,175.845,-107.384,169.415,44.303,158.360
C02595=1031.243,175.595,-107.361,169.412,44.305,158.360
C02596=1031.237,175.346,-107.338,169.409,44.307,158.360
C02597=1031.231,175.098,-107.314,169.405,44.309,158.360
C02598=1031.225,174.849,-107.292,169.403,44.310,158.360
C02599=1031.219,174.600,-107.269,169.399,44.313,158.360
C02600=1031.212,174.351,-107.245,169.396,44.314,158.360
C02601=1031.207,174.102,-107.222,169.394,44.316,158.360
C02602=1031.200,173.853,-107.200,169.390,44.317,158.360
C02603=1031.194,173.605,-107.176,169.387,44.319,158.360
C02604=1031.188,173.356,-107.153,169.384,44.321,158.361
C02605=1031.183,173.107,-107.131,169.381,44.322,158.361
C02606=1031.176,172.823,-107.105,169.377,44.325,158.361
C02607=1031.169,172.539,-107.078,169.374,44.327,158.361
C02608=1031.161,172.255,-107.052,169.370,44.329,158.361
C02609=1031.155,171.970,-107.026,169.367,44.331,158.361
C02610=1031.149,171.722,-107.003,169.364,44.332,158.361
C02611=1031.143,171.473,-106.980,169.360,44.334,158.361
C02612=1031.137,171.224,-106.958,169.358,44.336,158.361
C02613=1031.132,170.975,-106.935,169.355,44.337,158.361
C02614=1031.126,170.727,-106.911,169.351,44.340,158.361
C02615=1031.119,170.477,-106.888,169.349,44.341,158.361
C02616=1031.113,170.229,-106.865,169.345,44.343,158.361
C02617=1031.107,169.980,-106.842,169.342,44.345,158.362
C02618=1031.101,169.731,-106.819,169.340,44.347,158.362
C02619=1031.095,169.482,-106.797,169.336,44.348,158.362
C02620=1031.089,169.233,-106.774,169.333,44.350,158.362
C02621=1031.084,168.984,-106.752,169.331,44.352,158.362
C02622=1031.078,168.735,-106.729,169.327,44.354,158.362
C02623=1031.072,168.486,-106.707,169.324,44.355,158.362
C02624=1031.066,168.237,-106.684,169.322,44.357,158.362
C02625=1031.060,167.988,-106.661,169.318,44.359,158.362
C02626=1031.054,167.740,-106.638,169.315,44.361,158.362
C02627=1031.049,167.491,-106.615,169.313,44.362,158.362
C02628=1031.042,167.242,-106.592,169.309,44.364,158.362
C02629=1031.036,166.993,-106.569,169.306,44.366,158.362
C02630=1031.031,166.744,-106.547,169.304,44.367,158.362
C02631=1031.025,166.495,-106.524,169.300,44.369,158.363
C02632=1031.019,166.247,-106.501,169.297,44.371,158.363
C02633=1031.013,165.997,-106.479,169.295,44.373,158.363
C02634=1031.007,165.748,-106.456,169.291,44.375,158.363
C02635=1031.002,165.499,-106.433,169.288,44.377,158.363
C02636=1030.995,165.251,-106.411,169.286,44.378,158.363
C02637=1030.989,165.002,-106.388,169.282,44.380,158.363
C02638=1030.984,164.753,-106.365,169.279,44.382,158.363
C02639=1030.978,164.504,-106.343,169.277,44.383,158.363
C02640=1030.972,164.255,-106.320,169.273,44.385,158.363
C02641=1030.966,164.006,-106.297,169.270,44.387,158.363
C02642=1030.960,163.757,-106.274,169.268,44.388,158.363
C02643=1030.955,163.508,-106.251,169.265,44.390,158.364
C02644=1030.948,163.259,-106.230,169.262,44.392,158.364
C02645=1030.943,163.010,-106.207,169.259,44.394,158.364
C02646=1030.937,162.761,-106.184,169.256,44.396,158.364
C02647=1030.931,162.513,-106.162,169.253,44.398,158.364
C02648=1030.926,162.264,-106.140,169.250,44.399,158.364
C02649=1030.920,162.015,-106.117,169.247,44.401,158.364
C02650=1030.914,161.766,-106.094,169.245,44.403,158.364
C02651=1030.908,161.517,-106.072,169.241,44.404,158.364
C02652=1030.902,161.268,-106.049,169.238,44.406,158.364
C02653=1030.897,161.019,-106.026,169.236,44.408,158.364
C02654=1030.891,160.770,-106.003,169.233,44.409,158.364
C02655=1030.885,160.521,-105.982,169.229,44.412,158.364
C02656=1030.880,160.273,-105.959,169.227,44.413,158.365
C02657=1030.874,160.024,-105.936,169.224,44.415,158.365
C02658=1030.868,159.775,-105.915,169.221,44.417,158.365
C02659=1030.862,159.526,-105.892,169.218,44.419,158.365
C02660=1030.856,159.277,-105.870,169.215,44.421,158.365
C02661=1030.850,159.028,-105.847,169.213,44.423,158.365
C02662=1030.844,158.779,-105.825,169.209,44.424,158.365
C02663=1030.837,158.530,-105.803,169.206,44.426,158.365
C02664=1030.832,158.280,-105.781,169.204,44.428,158.365
C02665=1030.826,158.032,-105.758,169.201,44.430,158.366
C02666=1030.820,157.783,-105.737,169.197,44.432,158.366
C02667=1030.814,157.534,-105.716,169.195,44.434,158.366
C02668=1030.808,157.285,-105.693,169.192,44.436,158.366
C02669=1030.802,157.036,-105.671,169.189,44.438,158.366
C02670=1030.795,156.752,-105.645,169.186,44.440,158.366
C02671=1030.788,156.466,-105.620,169.183,44.442,158.366
C02672=1030.781,156.182,-105.595,169.179,44.444,158.366
C02673=1030.775,155.899,-105.570,169.175,44.446,158.366
C02674=1030.768,155.649,-105.548,169.173,44.448,158.367
C02675=1030.763,155.400,-105.526,169.170,44.450,158.367
C02676=1030.756,155.151,-105.504,169.168,44.452,158.367
C02677=1030.750,154.902,-105.482,169.164,44.454,158.367
C02678=1030.744,154.653,-105.460,169.161,44.456,158.367
C02679=1030.739,154.405,-105.438,169.159,44.458,158.367
C02680=1030.733,154.155,-105.416,169.156,44.460,158.367
C02681=1030.727,153.906,-105.395,169.153,44.462,158.367
C02682=1030.720,153.658,-105.372,169.150,44.464,158.368
C02683=1030.715,153.408,-105.350,169.148,44.466,158.368
C02684=1030.709,153.160,-105.329,169.145,44.468,158.368
C02685=1030.703,152.910,-105.307,169.141,44.470,158.368
C02686=1030.697,152.661,-105.285,169.139,44.472,158.368
C02687=1030.690,152.413,-105.263,169.136,44.474,158.368
C02688=1030.684,152.163,-105.241,169.132,44.475,158.368
C02689=1030.679,151.915,-105.220,169.130,44.477,158.368
C02690=1030.673,151.665,-105.198,169.127,44.479,158.368
C02691=1030.667,151.416,-105.176,169.125,44.481,158.369
C02692=1030.661,151.168,-105.154,169.121,44.483,158.369
C02693=1030.655,150.919,-105.133,169.119,44.485,158.369
C02694=1030.649,150.670,-105.111,169.116,44.487,158.369
C02695=1030.643,150.421,-105.089,169.113,44.489,158.369
C02696=1030.637,150.172,-105.068,169.111,44.491,158.369
C02697=1030.631,149.923,-105.047,169.107,44.493,158.369
C02698=1030.625,149.674,-105.024,169.105,44.495,158.369
C02699=1030.619,149.425,-105.002,169.102,44.497,158.370
C02700=1030.613,149.176,-104.980,169.100,44.499,158.370
C02701=1030.607,148.927,-104.959,169.096,44.501,158.370
C02702=1030.601,148.678,-104.937,169.093,44.503,158.370
C02703=1030.595,148.429,-104.916,169.091,44.505,158.370
C02704=1030.589,148.180,-104.894,169.088,44.507,158.370
C02705=1030.583,147.931,-104.873,169.086,44.509,158.370
C02706=1030.577,147.682,-104.851,169.082,44.511,158.371
C02707=1030.571,147.433,-104.830,169.080,44.513,158.371
C02708=1030.566,147.184,-104.808,169.077,44.515,158.371
C02709=1030.559,146.935,-104.787,169.074,44.516,158.371
C02710=1030.553,146.686,-104.765,169.072,44.518,158.371
C02711=1030.547,146.437,-104.743,169.068,44.521,158.371
C02712=1030.541,146.188,-104.722,169.066,44.522,158.371
C02713=1030.535,145.939,-104.701,169.063,44.524,158.371
C02714=1030.529,145.690,-104.679,169.061,44.527,158.372
C02715=1030.524,145.441,-104.658,169.057,44.529,158.372
C02716=1030.517,145.192,-104.636,169.055,44.531,158.372
C02717=1030.511,144.943,-104.614,169.052,44.533,158.372
C02718=1030.505,144.694,-104.594,169.049,44.535,158.372
C02719=1030.499,144.445,-104.573,169.047,44.537,158.372
C02720=1030.493,144.196,-104.551,169.043,44.539,158.372
C02721=1030.487,143.947,-104.530,169.041,44.541,158.373
C02722=1030.481,143.698,-104.508,169.038,44.543,158.373
C02723=1030.475,143.449,-104.487,169.036,44.545,158.373
C02724=1030.469,143.200,-104.465,169.033,44.547,158.373
C02725=1030.463,142.951,-104.445,169.030,44.549,158.373
C02726=1030.457,142.701,-104.423,169.027,44.551,158.373
C02727=1030.451,142.453,-104.402,169.025,44.553,158.374
C02728=1030.445,142.204,-104.380,169.022,44.555,158.374
C02729=1030.439,141.954,-104.359,169.019,44.557,158.374
C02730=1030.434,141.705,-104.338,169.016,44.559,158.374
C02731=1030.427,141.456,-104.317,169.013,44.561,158.374
C02732=1030.421,141.208,-104.296,169.011,44.563,158.374
C02733=1030.415,140.959,-104.274,169.008,44.565,158.374
C02734=1030.409,140.673,-104.250,169.005,44.568,158.375
C02735=1030.402,140.389,-104.226,169.002,44.570,158.375
C02736=1030.395,140.104,-104.202,168.999,44.572,158.375
C02737=1030.387,139.819,-104.177,168.996,44.575,158.375
C02738=1030.382,139.570,-104.157,168.993,44.577,158.375
C02739=1030.376,139.321,-104.135,168.990,44.579,158.375
C02740=1030.370,139.073,-104.114,168.988,44.581,158.375
C02741=1030.364,138.823,-104.093,168.985,44.583,158.376
C02742=1030.358,138.574,-104.071,168.982,44.584,158.376
C02743=1030.352,138.325,-104.051,168.980,44.586,158.376
C02744=1030.346,138.076,-104.030,168.976,44.589,158.376
C02745=1030.341,137.827,-104.008,168.974,44.591,158.376
C02746=1030.334,137.578,-103.988,168.971,44.593,158.376
C02747=1030.328,137.329,-103.967,168.969,44.595,158.377
C02748=1030.322,137.080,-103.945,168.966,44.597,158.377
C02749=1030.316,136.830,-103.925,168.964,44.599,158.377
C02750=1030.310,136.582,-103.904,168.960,44.602,158.377
C02751=1030.304,136.332,-103.883,168.958,44.604,158.377
C02752=1030.298,136.084,-103.862,168.955,44.606,158.377
C02753=1030.292,135.834,-103.841,168.953,44.608,158.377
C02754=1030.286,135.586,-103.820,168.950,44.609,158.378
C02755=1030.280,135.336,-103.799,168.948,44.612,158.378
C02756=1030.274,135.087,-103.778,168.944,44.614,158.378
C02757=1030.268,134.838,-103.758,168.942,44.616,158.378
C02758=1030.262,134.589,-103.737,168.939,44.618,158.378
C02759=1030.256,134.340,-103.716,168.936,44.620,158.378
C02760=1030.250,134.091,-103.695,168.934,44.622,158.378
C02761=1030.244,133.842,-103.675,168.932,44.625,158.379
C02762=1030.238,133.593,-103.653,168.929,44.626,158.379
C02763=1030.232,133.344,-103.633,168.926,44.628,158.379
C02764=1030.226,133.095,-103.612,168.923,44.631,158.379
C02765=1030.220,132.846,-103.591,168.920,44.633,158.379
C02766=1030.214,132.597,-103.570,168.918,44.635,158.380
C02767=1030.208,132.348,-103.549,168.915,44.637,158.380
C02768=1030.203,132.098,-103.529,168.913,44.639,158.380
C02769=1030.196,131.850,-103.508,168.910,44.641,158.380
C02770=1030.190,131.600,-103.487,168.908,44.643,158.380
C02771=1030.183,131.351,-103.466,168.905,44.645,158.380
C02772=1030.178,131.102,-103.446,168.902,44.648,158.380
C02773=1030.172,130.853,-103.425,168.899,44.650,158.381
C02774=1030.166,130.604,-103.404,168.897,44.652,158.381
C02775=1030.160,130.356,-103.384,168.894,44.653,158.381
C02776=1030.154,130.106,-103.363,168.892,44.656,158.381
C02777=1030.148,129.857,-103.343,168.889,44.658,158.381
C02778=1030.141,129.608,-103.322,168.887,44.660,158.381
C02779=1030.135,129.359,-103.302,168.883,44.663,158.382
C02780=1030.129,129.109,-103.281,168.881,44.665,158.382
C02781=1030.123,128.861,-103.261,168.878,44.667,158.382
C02782=1030.117,128.611,-103.241,168.876,44.669,158.382
C02783=1030.111,128.363,-103.220,168.873,44.671,158.382
C02784=1030.105,128.113,-103.199,168.871,44.673,158.383
C02785=1030.099,127.864,-103.179,168.867,44.676,158.383
C02786=1030.092,127.615,-103.159,168.865,44.678,158.383
C02787=1030.086,127.366,-103.139,168.862,44.680,158.383
C02788=1030.081,127.117,-103.118,168.860,44.682,158.383
C02789=1030.074,126.868,-103.098,168.857,44.684,158.383
C02790=1030.068,126.619,-103.078,168.855,44.686,158.384
C02791=1030.061,126.370,-103.057,168.852,44.689,158.384
C02792=1030.056,126.120,-103.037,168.850,44.691,158.384
C02793=1030.050,125.871,-103.016,168.846,44.693,158.384
C02794=1030.044,125.622,-102.996,168.844,44.696,158.384
C02795=1030.038,125.373,-102.976,168.841,44.698,158.384
C02796=1030.031,125.124,-102.955,168.839,44.700,158.385
C02797=1030.025,124.875,-102.935,168.836,44.702,158.385
C02798=1030.018,124.590,-102.912,168.833,44.704,158.385
C02799=1030.012,124.305,-102.889,168.830,44.707,158.385
C02800=1030.005,124.019,-102.866,168.827,44.710,158.386
C02801=1029.997,123.735,-102.843,168.825,44.712,158.386
C02802=1029.991,123.486,-102.823,168.822,44.714,158.386
C02803=1029.986,123.236,-102.802,168.820,44.716,158.386
C02804=1029.980,122.988,-102.782,168.816,44.718,158.386
C02805=1029.974,122.739,-102.762,168.814,44.720,158.386
C02806=1029.967,122.490,-102.741,168.811,44.723,158.387
C02807=1029.961,122.241,-102.720,168.809,44.725,158.387
C02808=1029.955,121.992,-102.701,168.806,44.727,158.387
C02809=1029.949,121.743,-102.680,168.804,44.729,158.387
C02810=1029.943,121.494,-102.660,168.801,44.731,158.387
C02811=1029.937,121.245,-102.640,168.799,44.733,158.387
C02812=1029.931,120.994,-102.620,168.796,44.735,158.388
C02813=1029.925,120.746,-102.600,168.794,44.738,158.388
C02814=1029.919,120.497,-102.580,168.791,44.740,158.388
C02815=1029.913,120.247,-102.560,168.789,44.742,158.388
C02816=1029.907,119.998,-102.539,168.786,44.744,158.388
C02817=1029.901,119.749,-102.519,168.783,44.747,158.388
C02818=1029.895,119.501,-102.499,168.780,44.749,158.389
C02819=1029.889,119.251,-102.479,168.778,44.751,158.389
C02820=1029.883,119.002,-102.459,168.775,44.753,158.389
C02821=1029.878,118.753,-102.439,168.773,44.755,158.389
C02822=1029.872,118.504,-102.419,168.770,44.757,158.389
C02823=1029.865,118.255,-102.398,168.768,44.759,158.389
C02824=1029.859,118.006,-102.378,168.765,44.762,158.390
C02825=1029.853,117.757,-102.358,168.763,44.764,158.390
C02826=1029.848,117.507,-102.338,168.760,44.765,158.390
C02827=1029.841,117.258,-102.318,168.758,44.767,158.390
C02828=1029.835,117.009,-102.298,168.755,44.770,158.390
C02829=1029.829,116.760,-102.278,168.753,44.772,158.390
C02830=1029.823,116.511,-102.258,168.750,44.774,158.391
C02831=1029.818,116.262,-102.237,168.748,44.776,158.391
C02832=1029.812,116.012,-102.218,168.745,44.779,158.391
C02833=1029.806,115.763,-102.198,168.743,44.780,158.391
C02834=1029.800,115.515,-102.178,168.740,44.782,158.391
C02835=1029.794,115.266,-102.158,168.737,44.784,158.391
C02836=1029.788,115.016,-102.137,168.735,44.787,158.392
C02837=1029.782,114.767,-102.117,168.733,44.789,158.392
C02838=1029.776,114.518,-102.098,168.730,44.791,158.392
C02839=1029.770,114.269,-102.078,168.727,44.793,158.392
C02840=1029.764,114.020,-102.058,168.725,44.796,158.392
C02841=1029.758,113.771,-102.038,168.723,44.797,158.393
C02842=1029.753,113.521,-102.018,168.720,44.799,158.393
C02843=1029.747,113.272,-101.998,168.717,44.801,158.393
C02844=1029.741,113.023,-101.978,168.715,44.803,158.393
C02845=1029.735,112.774,-101.959,168.713,44.806,158.393
C02846=1029.729,112.525,-101.939,168.710,44.808,158.393
C02847=1029.723,112.275,-101.919,168.708,44.811,158.394
C02848=1029.717,112.026,-101.899,168.704,44.813,158.394
C02849=1029.711,111.777,-101.879,168.702,44.815,158.394
C02850=1029.705,111.528,-101.859,168.699,44.817,158.394
C02851=1029.699,111.279,-101.840,168.697,44.819,158.394
C02852=1029.693,111.030,-101.821,168.694,44.821,158.394
C02853=1029.686,110.780,-101.801,168.692,44.824,158.395
C02854=1029.680,110.531,-101.781,168.689,44.826,158.395
C02855=1029.674,110.283,-101.761,168.687,44.828,158.395
C02856=1029.669,110.033,-101.742,168.684,44.830,158.395
C02857=1029.663,109.784,-101.722,168.682,44.832,158.395
C02858=1029.656,109.534,-101.702,168.679,44.835,158.396
C02859=1029.650,109.286,-101.683,168.677,44.837,158.396
C02860=1029.644,109.036,-101.664,168.675,44.840,158.396
C02861=1029.638,108.788,-101.644,168.672,44.841,158.396
C02862=1029.631,108.503,-101.622,168.669,44.844,158.396
C02863=1029.624,108.217,-101.600,168.666,44.847,158.397
C02864=1029.617,107.932,-101.578,168.663,44.849,158.397
C02865=1029.610,107.647,-101.556,168.660,44.852,158.397
C02866=1029.604,107.398,-101.536,168.658,44.854,158.397
C02867=1029.598,107.149,-101.516,168.656,44.856,158.397
C02868=1029.591,106.900,-101.497,168.653,44.858,158.398
C02869=1029.585,106.650,-101.477,168.651,44.861,158.398
C02870=1029.579,106.401,-101.458,168.648,44.863,158.398
C02871=1029.574,106.152,-101.438,168.646,44.866,158.398
C02872=1029.567,105.903,-101.420,168.643,44.867,158.398
C02873=1029.561,105.654,-101.400,168.641,44.869,158.399
C02874=1029.555,105.404,-101.380,168.638,44.872,158.399
C02875=1029.549,105.156,-101.361,168.636,44.874,158.399
C02876=1029.543,104.906,-101.342,168.633,44.877,158.399
C02877=1029.537,104.657,-101.323,168.630,44.879,158.399
C02878=1029.531,104.408,-101.303,168.627,44.881,158.399
C02879=1029.525,104.159,-101.284,168.625,44.883,158.400
C02880=1029.519,103.909,-101.264,168.622,44.885,158.400
C02881=1029.513,103.660,-101.244,168.620,44.887,158.400
C02882=1029.507,103.411,-101.225,168.618,44.890,158.400
C02883=1029.500,103.162,-101.206,168.615,44.892,158.400
C02884=1029.494,102.913,-101.187,168.613,44.895,158.401
C02885=1029.489,102.663,-101.167,168.610,44.897,158.401
C02886=1029.482,102.414,-101.149,168.608,44.898,158.401
C02887=1029.476,102.165,-101.129,168.605,44.901,158.401
C02888=1029.471,101.916,-101.109,168.603,44.903,158.401
C02889=1029.465,101.666,-101.090,168.600,44.905,158.401
C02890=1029.459,101.417,-101.072,168.598,44.908,158.402
C02891=1029.453,101.169,-101.052,168.595,44.910,158.402
C02892=1029.447,100.919,-101.032,168.593,44.912,158.402
C02893=1029.440,100.670,-101.014,168.590,44.914,158.402
C02894=1029.435,100.421,-100.994,168.588,44.916,158.402
C02895=1029.429,100.172,-100.974,168.585,44.919,158.403
C02896=1029.423,99.922,-100.955,168.583,44.921,158.403
C02897=1029.417,99.673,-100.937,168.580,44.923,158.403
C02898=1029.410,99.424,-100.918,168.578,44.925,158.403
C02899=1029.405,99.175,-100.899,168.575,44.927,158.403
C02900=1029.398,98.926,-100.880,168.573,44.930,158.404
C02901=1029.392,98.676,-100.861,168.571,44.932,158.404
C02902=1029.386,98.428,-100.841,168.568,44.935,158.404
C02903=1029.380,98.178,-100.822,168.566,44.937,158.404
C02904=1029.374,97.929,-100.804,168.563,44.939,158.404
C02905=1029.368,97.680,-100.784,168.561,44.941,158.405
C02906=1029.361,97.430,-100.766,168.559,44.944,158.405
C02907=1029.355,97.181,-100.747,168.556,44.946,158.405
C02908=1029.349,96.932,-100.728,168.554,44.948,158.405
C02909=1029.343,96.683,-100.709,168.551,44.950,158.405
C02910=1029.337,96.433,-100.690,168.549,44.953,158.406
C02911=1029.331,96.184,-100.671,168.546,44.955,158.406
C02912=1029.325,95.935,-100.652,168.544,44.957,158.406
C02913=1029.319,95.686,-100.633,168.541,44.960,158.406
C02914=1029.312,95.437,-100.615,168.539,44.962,158.406
C02915=1029.307,95.187,-100.595,168.536,44.964,158.407
C02916=1029.300,94.938,-100.577,168.534,44.966,158.407
C02917=1029.294,94.689,-100.558,168.532,44.969,158.407
C02918=1029.288,94.439,-100.539,168.529,44.971,158.407
C02919=1029.282,94.190,-100.520,168.527,44.973,158.407
C02920=1029.276,93.941,-100.501,168.524,44.975,158.407
C02921=1029.270,93.692,-100.482,168.522,44.977,158.408
C02922=1029.264,93.443,-100.463,168.519,44.980,158.408
C02923=1029.258,93.194,-100.445,168.517,44.982,158.408
C02924=1029.252,92.945,-100.426,168.514,44.985,158.408
C02925=1029.246,92.695,-100.407,168.512,44.987,158.408
C02926=1029.238,92.386,-100.384,168.509,44.989,158.409
C02927=1029.231,92.078,-100.360,168.506,44.992,158.409
C02928=1029.223,91.770,-100.337,168.503,44.995,158.409
C02929=1029.216,91.461,-100.314,168.500,44.998,158.409
C02930=1029.210,91.211,-100.295,168.497,45.000,158.409
C02931=1029.204,90.962,-100.276,168.495,45.002,158.410
C02932=1029.197,90.713,-100.257,168.492,45.004,158.410
C02933=1029.192,90.463,-100.238,168.490,45.007,158.410
C02934=1029.185,90.214,-100.219,168.487,45.009,158.410
C02935=1029.180,89.965,-100.201,168.485,45.011,158.410
C02936=1029.174,89.716,-100.183,168.482,45.014,158.411
C02937=1029.168,89.467,-100.164,168.480,45.016,158.411
C02938=1029.161,89.218,-100.145,168.478,45.018,158.411
C02939=1029.155,88.968,-100.127,168.475,45.020,158.411
C02940=1029.149,88.718,-100.108,168.473,45.023,158.411
C02941=1029.143,88.469,-100.090,168.470,45.026,158.412
C02942=1029.136,88.220,-100.071,168.468,45.028,158.412
C02943=1029.130,87.970,-100.053,168.465,45.030,158.412
C02944=1029.125,87.722,-100.035,168.463,45.032,158.412
C02945=1029.118,87.473,-100.016,168.461,45.035,158.413
C02946=1029.112,87.224,-99.997,168.458,45.037,158.413
C02947=1029.106,86.974,-99.979,168.456,45.039,158.413
C02948=1029.100,86.725,-99.960,168.453,45.041,158.413
C02949=1029.093,86.476,-99.942,168.451,45.044,158.413
C02950=1029.087,86.226,-99.924,168.448,45.046,158.413
C02951=1029.081,85.977,-99.905,168.446,45.049,158.414
C02952=1029.075,85.728,-99.887,168.443,45.051,158.414
C02953=1029.069,85.478,-99.869,168.441,45.053,158.414
C02954=1029.063,85.241,-99.851,168.439,45.055,158.414
C02955=1029.057,85.004,-99.834,168.436,45.058,158.415
C02956=1029.051,84.766,-99.816,168.435,45.060,158.415
C02957=1029.045,84.529,-99.798,168.432,45.062,158.415
C02958=1029.039,84.291,-99.781,168.430,45.064,158.415
C02959=1029.034,84.054,-99.764,168.427,45.066,158.415
C02960=1029.028,83.817,-99.746,168.425,45.068,158.415
C02961=1029.023,83.579,-99.728,168.422,45.071,158.416
C02962=1029.016,83.330,-99.710,168.420,45.073,158.416
C02963=1029.010,83.080,-99.692,168.418,45.076,158.416
C02964=1029.004,82.831,-99.673,168.415,45.078,158.416
C02965=1028.998,82.582,-99.656,168.413,45.080,158.416
C02966=1028.992,82.333,-99.637,168.410,45.082,158.417
C02967=1028.986,82.083,-99.619,168.408,45.085,158.417
C02968=1028.979,81.834,-99.600,168.405,45.087,158.417
C02969=1028.973,81.586,-99.582,168.403,45.089,158.417
C02970=1028.967,81.336,-99.564,168.400,45.091,158.417
C02971=1028.962,81.087,-99.545,168.399,45.093,158.418
C02972=1028.955,80.837,-99.527,168.397,45.096,158.418
C02973=1028.950,80.589,-99.509,168.394,45.098,158.418
C02974=1028.943,80.339,-99.491,168.392,45.101,158.418
C02975=1028.937,80.090,-99.472,168.389,45.102,158.418
C02976=1028.931,79.840,-99.454,168.387,45.105,158.419
C02977=1028.925,79.591,-99.436,168.384,45.107,158.419
C02978=1028.919,79.342,-99.418,168.382,45.109,158.419
C02979=1028.913,79.093,-99.399,168.379,45.112,158.419
C02980=1028.907,78.844,-99.382,168.377,45.114,158.419
C02981=1028.901,78.594,-99.363,168.375,45.116,158.420
C02982=1028.895,78.345,-99.345,168.372,45.118,158.420
C02983=1028.888,78.096,-99.326,168.370,45.121,158.420
C02984=1028.883,77.846,-99.308,168.367,45.123,158.420
C02985=1028.876,77.597,-99.291,168.365,45.125,158.420
C02986=1028.870,77.348,-99.272,168.362,45.128,158.420
C02987=1028.865,77.099,-99.255,168.360,45.130,158.421
C02988=1028.858,76.850,-99.236,168.357,45.132,158.421
C02989=1028.852,76.600,-99.218,168.355,45.134,158.421
C02990=1028.845,76.314,-99.197,168.352,45.137,158.421
C02991=1028.838,76.030,-99.177,168.349,45.140,158.421
C02992=1028.831,75.745,-99.156,168.347,45.142,158.422
C02993=1028.824,75.459,-99.137,168.344,45.145,158.422
C02994=1028.818,75.210,-99.118,168.341,45.148,158.422
C02995=1028.812,74.961,-99.100,168.339,45.150,158.422
C02996=1028.806,74.711,-99.082,168.336,45.153,158.423
C02997=1028.800,74.462,-99.064,168.334,45.155,158.423
C02998=1028.793,74.213,-99.047,168.331,45.157,158.423
C02999=1028.787,73.963,-99.029,168.329,45.159,158.423
C03000=1028.781,73.714,-99.011,168.327,45.162,158.423
C03001=1028.775,73.465,-98.993,168.324,45.164,158.424
C03002=1028.769,73.215,-98.975,168.322,45.167,158.424
C03003=1028.763,72.967,-98.958,168.319,45.169,158.424
C03004=1028.756,72.717,-98.940,168.317,45.171,158.424
C03005=1028.750,72.468,-98.921,168.314,45.173,158.424
C03006=1028.745,72.219,-98.904,168.312,45.176,158.425
C03007=1028.738,71.969,-98.886,168.309,45.178,158.425
C03008=1028.732,71.719,-98.868,168.307,45.181,158.425
C03009=1028.726,71.470,-98.851,168.305,45.183,158.425
C03010=1028.720,71.221,-98.832,168.302,45.185,158.425
C03011=1028.714,70.972,-98.815,168.300,45.187,158.425
C03012=1028.707,70.723,-98.797,168.298,45.190,158.426
C03013=1028.701,70.473,-98.779,168.296,45.192,158.426
C03014=1028.696,70.224,-98.762,168.294,45.194,158.426
C03015=1028.689,69.974,-98.744,168.291,45.196,158.426
C03016=1028.683,69.726,-98.727,168.289,45.199,158.427
C03017=1028.677,69.476,-98.708,168.286,45.201,158.427
C03018=1028.671,69.227,-98.690,168.284,45.203,158.427
C03019=1028.665,68.978,-98.673,168.281,45.206,158.427
C03020=1028.658,68.728,-98.655,168.279,45.208,158.427
C03021=1028.653,68.479,-98.638,168.276,45.210,158.427
C03022=1028.647,68.229,-98.620,168.274,45.213,158.428
C03023=1028.640,67.980,-98.602,168.272,45.215,158.428
C03024=1028.634,67.731,-98.585,168.269,45.218,158.428
C03025=1028.627,67.482,-98.568,168.267,45.220,158.428
C03026=1028.622,67.233,-98.550,168.264,45.222,158.429
C03027=1028.616,66.983,-98.532,168.262,45.224,158.429
C03028=1028.610,66.734,-98.515,168.260,45.227,158.429
C03029=1028.603,66.484,-98.497,168.257,45.229,158.429
C03030=1028.597,66.235,-98.479,168.255,45.232,158.429
C03031=1028.591,65.986,-98.462,168.252,45.234,158.429
C03032=1028.585,65.736,-98.444,168.250,45.236,158.430
C03033=1028.579,65.487,-98.427,168.247,45.238,158.430
C03034=1028.573,65.238,-98.409,168.245,45.241,158.430
C03035=1028.566,64.989,-98.392,168.242,45.243,158.430
C03036=1028.560,64.739,-98.374,168.240,45.246,158.430
C03037=1028.554,64.490,-98.358,168.238,45.248,158.431
C03038=1028.548,64.241,-98.340,168.235,45.250,158.431
C03039=1028.542,63.992,-98.322,168.233,45.252,158.431
C03040=1028.535,63.742,-98.305,168.230,45.255,158.431
C03041=1028.530,63.493,-98.287,168.228,45.257,158.431
C03042=1028.523,63.243,-98.270,168.226,45.260,158.432
C03043=1028.517,62.994,-98.254,168.223,45.262,158.432
C03044=1028.511,62.745,-98.236,168.221,45.264,158.432
C03045=1028.504,62.495,-98.218,168.218,45.267,158.432
C03046=1028.498,62.247,-98.201,168.216,45.270,158.433
C03047=1028.491,61.996,-98.185,168.213,45.272,158.433
C03048=1028.486,61.747,-98.167,168.210,45.274,158.433
C03049=1028.479,61.498,-98.150,168.208,45.277,158.433
C03050=1028.473,61.249,-98.133,168.205,45.279,158.433
C03051=1028.467,60.999,-98.116,168.203,45.282,158.434
C03052=1028.461,60.750,-98.099,168.201,45.285,158.434
C03053=1028.454,60.501,-98.081,168.198,45.287,158.434
C03054=1028.447,60.216,-98.062,168.196,45.289,158.434
C03055=1028.440,59.930,-98.042,168.193,45.292,158.434
C03056=1028.433,59.645,-98.023,168.190,45.295,158.435
C03057=1028.425,59.360,-98.003,168.187,45.298,158.435
C03058=1028.419,59.110,-97.986,168.185,45.300,158.435
C03059=1028.412,58.861,-97.969,168.182,45.303,158.435
C03060=1028.407,58.612,-97.951,168.180,45.305,158.436
C03061=1028.400,58.362,-97.935,168.178,45.308,158.436
C03062=1028.394,58.113,-97.918,168.175,45.310,158.436
C03063=1028.387,57.864,-97.901,168.173,45.312,158.436
C03064=1028.382,57.614,-97.884,168.170,45.315,158.436
C03065=1028.375,57.365,-97.866,168.168,45.317,158.437
C03066=1028.369,57.116,-97.849,168.166,45.320,158.437
C03067=1028.362,56.866,-97.833,168.163,45.322,158.437
C03068=1028.357,56.617,-97.815,168.161,45.324,158.437
C03069=1028.351,56.367,-97.799,168.158,45.327,158.437
C03070=1028.344,56.118,-97.782,168.156,45.329,158.438
C03071=1028.338,55.869,-97.765,168.154,45.332,158.438
C03072=1028.332,55.619,-97.747,168.151,45.334,158.438
C03073=1028.326,55.370,-97.730,168.149,45.336,158.438
C03074=1028.319,55.120,-97.714,168.146,45.338,158.438
C03075=1028.313,54.871,-97.697,168.144,45.341,158.439
C03076=1028.307,54.622,-97.679,168.142,45.344,158.439
C03077=1028.301,54.372,-97.663,168.139,45.346,158.439
C03078=1028.295,54.124,-97.646,168.137,45.348,158.439
C03079=1028.288,53.874,-97.629,168.134,45.350,158.439
C03080=1028.283,53.624,-97.612,168.132,45.353,158.440
C03081=1028.277,53.375,-97.595,168.129,45.355,158.440
C03082=1028.270,53.126,-97.578,168.127,45.358,158.440
C03083=1028.264,52.876,-97.562,168.124,45.360,158.440
C03084=1028.258,52.627,-97.544,168.122,45.363,158.440
C03085=1028.251,52.378,-97.527,168.120,45.365,158.441
C03086=1028.245,52.129,-97.510,168.117,45.367,158.441
C03087=1028.239,51.880,-97.494,168.115,45.370,158.441
C03088=1028.233,51.630,-97.477,168.112,45.372,158.441
C03089=1028.227,51.381,-97.459,168.110,45.375,158.441
C03090=1028.221,51.131,-97.443,168.108,45.377,158.442
C03091=1028.215,50.881,-97.426,168.105,45.379,158.442
C03092=1028.208,50.633,-97.409,168.103,45.381,158.442
C03093=1028.203,50.383,-97.393,168.100,45.384,158.442
C03094=1028.196,50.133,-97.375,168.098,45.386,158.442
C03095=1028.190,49.884,-97.359,168.096,45.389,158.443
C03096=1028.184,49.635,-97.342,168.093,45.391,158.443
C03097=1028.178,49.385,-97.325,168.091,45.393,158.443
C03098=1028.172,49.136,-97.308,168.088,45.395,158.443
C03099=1028.166,48.887,-97.292,168.086,45.397,158.443
C03100=1028.159,48.637,-97.275,168.083,45.400,158.443
C03101=1028.153,48.388,-97.258,168.081,45.402,158.444
C03102=1028.148,48.139,-97.241,168.079,45.405,158.444
C03103=1028.142,47.890,-97.224,168.076,45.407,158.444
C03104=1028.135,47.640,-97.208,168.074,45.409,158.444
C03105=1028.129,47.390,-97.191,168.071,45.411,158.444
C03106=1028.123,47.142,-97.174,168.069,45.414,158.445
C03107=1028.118,46.892,-97.157,168.066,45.416,158.445
C03108=1028.111,46.643,-97.140,168.064,45.419,158.445
C03109=1028.105,46.393,-97.124,168.061,45.421,158.445
C03110=1028.099,46.144,-97.108,168.059,45.423,158.445
C03111=1028.093,45.895,-97.091,168.057,45.426,158.445
C03112=1028.087,45.645,-97.073,168.054,45.428,158.446
C03113=1028.081,45.395,-97.057,168.052,45.430,158.446
C03114=1028.075,45.147,-97.040,168.049,45.432,158.446
C03115=1028.069,44.897,-97.024,168.047,45.434,158.446
C03116=1028.062,44.647,-97.007,168.044,45.437,158.446
C03117=1028.057,44.398,-96.990,168.042,45.439,158.446
C03118=1028.050,44.113,-96.972,168.038,45.442,158.447
C03119=1028.042,43.827,-96.952,168.036,45.445,158.447
C03120=1028.036,43.541,-96.933,168.034,45.447,158.447
C03121=1028.029,43.256,-96.914,168.030,45.450,158.447
C03122=1028.023,43.006,-96.897,168.028,45.452,158.447
C03123=1028.017,42.757,-96.881,168.025,45.454,158.448
C03124=1028.011,42.507,-96.865,168.023,45.457,158.448
C03125=1028.005,42.258,-96.848,168.021,45.459,158.448
C03126=1027.998,42.010,-96.832,168.018,45.462,158.448
C03127=1027.992,41.760,-96.815,168.016,45.464,158.448
C03128=1027.986,41.510,-96.799,168.014,45.466,158.449
C03129=1027.980,41.261,-96.783,168.011,45.468,158.449
C03130=1027.974,41.011,-96.767,168.009,45.471,158.449
C03131=1027.968,40.762,-96.750,168.006,45.473,158.449
C03132=1027.962,40.512,-96.734,168.004,45.476,158.449
C03133=1027.956,40.263,-96.717,168.001,45.478,158.449
C03134=1027.950,40.013,-96.701,167.999,45.480,158.450
C03135=1027.943,39.765,-96.684,167.996,45.482,158.450
C03136=1027.937,39.515,-96.668,167.994,45.485,158.450
C03137=1027.931,39.265,-96.651,167.992,45.487,158.450
C03138=1027.925,39.016,-96.635,167.989,45.490,158.450
C03139=1027.918,38.767,-96.619,167.987,45.492,158.451
C03140=1027.912,38.518,-96.603,167.984,45.495,158.451
C03141=1027.906,38.268,-96.587,167.982,45.497,158.451
C03142=1027.900,38.019,-96.571,167.980,45.499,158.451
C03143=1027.894,37.769,-96.554,167.977,45.501,158.451
C03144=1027.888,37.519,-96.538,167.975,45.504,158.452
C03145=1027.882,37.270,-96.521,167.972,45.506,158.452
C03146=1027.876,37.021,-96.505,167.970,45.509,158.452
C03147=1027.870,36.771,-96.489,167.967,45.511,158.452
C03148=1027.863,36.522,-96.473,167.964,45.514,158.452
C03149=1027.857,36.273,-96.457,167.962,45.516,158.452
C03150=1027.851,36.024,-96.441,167.959,45.518,158.453
C03151=1027.844,35.774,-96.425,167.957,45.521,158.453
C03152=1027.838,35.525,-96.408,167.954,45.523,158.453
C03153=1027.833,35.275,-96.393,167.952,45.526,158.453
C03154=1027.826,35.026,-96.377,167.950,45.529,158.453
C03155=1027.820,34.776,-96.361,167.947,45.531,158.454
C03156=1027.814,34.527,-96.345,167.945,45.533,158.454
C03157=1027.807,34.278,-96.329,167.942,45.535,158.454
C03158=1027.801,34.028,-96.313,167.940,45.538,158.454
C03159=1027.795,33.779,-96.297,167.938,45.541,158.454
C03160=1027.789,33.529,-96.282,167.935,45.543,158.455
C03161=1027.782,33.279,-96.265,167.933,45.545,158.455
C03162=1027.776,33.030,-96.249,167.929,45.548,158.455
C03163=1027.770,32.781,-96.233,167.927,45.550,158.455
C03164=1027.764,32.532,-96.217,167.925,45.552,158.455
C03165=1027.758,32.282,-96.201,167.922,45.555,158.456
C03166=1027.751,32.033,-96.186,167.920,45.557,158.456
C03167=1027.746,31.783,-96.169,167.917,45.560,158.456
C03168=1027.740,31.534,-96.153,167.915,45.562,158.456
C03169=1027.733,31.285,-96.137,167.913,45.564,158.456
C03170=1027.727,31.036,-96.121,167.910,45.567,158.457
C03171=1027.721,30.786,-96.106,167.908,45.569,158.457
C03172=1027.715,30.537,-96.090,167.906,45.572,158.457
C03173=1027.709,30.287,-96.074,167.903,45.574,158.457
C03174=1027.703,30.038,-96.058,167.901,45.577,158.457
C03175=1027.696,29.788,-96.043,167.898,45.579,158.457
C03176=1027.690,29.539,-96.026,167.896,45.581,158.458
C03177=1027.684,29.290,-96.010,167.893,45.583,158.458
C03178=1027.678,29.040,-95.995,167.891,45.586,158.458
C03179=1027.672,28.791,-95.979,167.887,45.588,158.458
C03180=1027.666,28.541,-95.963,167.885,45.591,158.458
C03181=1027.659,28.292,-95.947,167.883,45.593,158.458
C03182=1027.652,28.005,-95.929,167.880,45.596,158.459
C03183=1027.646,27.720,-95.911,167.877,45.599,158.459
C03184=1027.638,27.435,-95.893,167.875,45.601,158.459
C03185=1027.631,27.149,-95.875,167.871,45.604,158.459
C03186=1027.625,26.899,-95.860,167.869,45.606,158.459
C03187=1027.619,26.650,-95.844,167.867,45.609,158.460
C03188=1027.612,26.401,-95.828,167.864,45.612,158.460
C03189=1027.607,26.151,-95.812,167.862,45.614,158.460
C03190=1027.600,25.902,-95.797,167.859,45.617,158.460
C03191=1027.594,25.652,-95.781,167.857,45.619,158.460
C03192=1027.588,25.403,-95.766,167.855,45.621,158.461
C03193=1027.582,25.153,-95.750,167.851,45.624,158.461
C03194=1027.575,24.904,-95.734,167.849,45.626,158.461
C03195=1027.569,24.654,-95.719,167.846,45.629,158.461
C03196=1027.563,24.405,-95.703,167.844,45.631,158.461
C03197=1027.556,24.155,-95.688,167.842,45.634,158.462
C03198=1027.551,23.906,-95.672,167.839,45.636,158.462
C03199=1027.544,23.656,-95.657,167.837,45.638,158.462
C03200=1027.538,23.407,-95.641,167.835,45.641,158.462
C03201=1027.532,23.158,-95.626,167.832,45.643,158.462
C03202=1027.526,22.909,-95.610,167.830,45.646,158.463
C03203=1027.520,22.659,-95.595,167.826,45.648,158.463
C03204=1027.513,22.410,-95.579,167.824,45.651,158.463
C03205=1027.508,22.160,-95.564,167.821,45.653,158.463
C03206=1027.501,21.911,-95.548,167.819,45.656,158.463
C03207=1027.495,21.661,-95.533,167.816,45.658,158.463
C03208=1027.489,21.412,-95.517,167.814,45.660,158.464
C03209=1027.482,21.162,-95.502,167.812,45.662,158.464
C03210=1027.477,20.912,-95.486,167.809,45.665,158.464
C03211=1027.470,20.663,-95.471,167.807,45.667,158.464
C03212=1027.464,20.414,-95.456,167.804,45.670,158.464
C03213=1027.458,20.165,-95.440,167.801,45.672,158.464
C03214=1027.452,19.915,-95.425,167.799,45.675,158.465
C03215=1027.446,19.665,-95.409,167.796,45.678,158.465
C03216=1027.440,19.416,-95.394,167.794,45.680,158.465
C03217=1027.433,19.167,-95.379,167.792,45.682,158.465
C03218=1027.427,18.917,-95.364,167.789,45.684,158.465
C03219=1027.421,18.668,-95.348,167.787,45.687,158.466
C03220=1027.415,18.419,-95.333,167.784,45.689,158.466
C03221=1027.409,18.169,-95.318,167.781,45.692,158.466
C03222=1027.402,17.920,-95.302,167.779,45.695,158.466
C03223=1027.396,17.670,-95.287,167.776,45.697,158.466
C03224=1027.390,17.420,-95.272,167.774,45.699,158.466
C03225=1027.384,17.171,-95.257,167.771,45.701,158.467
C03226=1027.377,16.922,-95.241,167.769,45.704,158.467
C03227=1027.372,16.672,-95.226,167.766,45.706,158.467
C03228=1027.365,16.423,-95.211,167.764,45.709,158.467
C03229=1027.359,16.173,-95.196,167.761,45.711,158.467
C03230=1027.352,15.924,-95.181,167.758,45.714,158.467
C03231=1027.347,15.674,-95.165,167.756,45.717,158.468
C03232=1027.341,15.425,-95.150,167.753,45.719,158.468
C03233=1027.335,15.175,-95.135,167.751,45.721,158.468
C03234=1027.328,14.926,-95.121,167.749,45.723,158.468
C03235=1027.322,14.676,-95.104,167.746,45.726,158.468
C03236=1027.316,14.427,-95.089,167.744,45.728,158.469
C03237=1027.310,14.178,-95.075,167.740,45.731,158.469
C03238=1027.304,13.928,-95.060,167.738,45.733,158.469
C03239=1027.298,13.678,-95.044,167.736,45.736,158.469
C03240=1027.292,13.429,-95.029,167.733,45.738,158.469
C03241=1027.285,13.179,-95.014,167.731,45.741,158.469
C03242=1027.279,12.929,-94.999,167.729,45.743,158.470
C03243=1027.273,12.681,-94.984,167.725,45.746,158.470
C03244=1027.266,12.431,-94.969,167.723,45.748,158.470
C03245=1027.260,12.182,-94.954,167.720,45.751,158.470
C03246=1027.252,11.897,-94.938,167.717,45.754,158.470
C03247=1027.246,11.612,-94.921,167.715,45.757,158.471
C03248=1027.238,11.328,-94.904,167.711,45.760,158.471
C03249=1027.232,11.044,-94.887,167.709,45.762,158.471
C03250=1027.225,10.795,-94.872,167.706,45.765,158.471
C03251=1027.219,10.545,-94.857,167.703,45.767,158.471
C03252=1027.213,10.295,-94.842,167.701,45.770,158.472
C03253=1027.207,10.046,-94.828,167.699,45.773,158.472
C03254=1027.200,9.797,-94.813,167.696,45.775,158.472
C03255=1027.194,9.547,-94.798,167.693,45.778,158.472
C03256=1027.188,9.297,-94.783,167.690,45.780,158.472
C03257=1027.182,9.048,-94.768,167.688,45.783,158.473
C03258=1027.175,8.799,-94.753,167.686,45.785,158.473
C03259=1027.168,8.549,-94.739,167.683,45.787,158.473
C03260=1027.162,8.300,-94.724,167.680,45.790,158.473
C03261=1027.156,8.051,-94.710,167.678,45.793,158.473
C03262=1027.150,7.801,-94.695,167.675,45.795,158.473
C03263=1027.144,7.551,-94.680,167.673,45.798,158.474
C03264=1027.138,7.302,-94.666,167.670,45.800,158.474
C03265=1027.132,7.052,-94.651,167.668,45.803,158.474
C03266=1027.125,6.803,-94.636,167.664,45.805,158.474
C03267=1027.119,6.554,-94.621,167.662,45.808,158.474
C03268=1027.113,6.304,-94.606,167.660,45.810,158.475
C03269=1027.107,6.054,-94.591,167.657,45.812,158.475
C03270=1027.101,5.805,-94.577,167.655,45.815,158.475
C03271=1027.095,5.555,-94.563,167.652,45.817,158.475
C03272=1027.088,5.305,-94.548,167.649,45.820,158.475
C03273=1027.083,5.056,-94.533,167.647,45.823,158.475
C03274=1027.076,4.807,-94.518,167.644,45.825,158.476
C03275=1027.070,4.557,-94.503,167.642,45.828,158.476
C03276=1027.064,4.308,-94.489,167.640,45.830,158.476
C03277=1027.058,4.058,-94.474,167.636,45.833,158.476
C03278=1027.051,3.809,-94.460,167.634,45.835,158.476
C03279=1027.045,3.560,-94.446,167.632,45.837,158.476
C03280=1027.039,3.310,-94.431,167.629,45.839,158.477
C03281=1027.033,3.061,-94.416,167.627,45.842,158.477
C03282=1027.027,2.811,-94.402,167.623,45.844,158.477
C03283=1027.020,2.561,-94.387,167.621,45.847,158.477
C03284=1027.015,2.312,-94.372,167.619,45.850,158.477
C03285=1027.008,2.062,-94.357,167.616,45.852,158.477
C03286=1027.003,1.813,-94.343,167.614,45.855,158.478
C03287=1026.996,1.563,-94.328,167.611,45.857,158.478
C03288=1026.991,1.314,-94.314,167.608,45.860,158.478
C03289=1026.985,1.064,-94.300,167.605,45.862,158.478
C03290=1026.978,0.814,-94.285,167.603,45.865,158.478
C03291=1026.972,0.565,-94.270,167.601,45.867,158.478
C03292=1026.965,0.316,-94.256,167.598,45.869,158.479
C03293=1026.960,0.066,-94.242,167.595,45.872,158.479
C03294=1026.953,-0.183,-94.227,167.592,45.874,158.479
C03295=1026.948,-0.432,-94.212,167.590,45.876,158.479
C03296=1026.942,-0.682,-94.198,167.588,45.879,158.479
C03297=1026.936,-0.931,-94.184,167.585,45.881,158.479
C03298=1026.929,-1.181,-94.169,167.583,45.883,158.479
C03299=1026.924,-1.431,-94.155,167.579,45.886,158.480
C03300=1026.918,-1.680,-94.140,167.577,45.888,158.480
C03301=1026.912,-1.929,-94.125,167.574,45.891,158.480
C03302=1026.906,-2.179,-94.111,167.572,45.893,158.480
C03303=1026.899,-2.428,-94.097,167.570,45.896,158.480
C03304=1026.893,-2.678,-94.083,167.567,45.898,158.480
C03305=1026.887,-2.927,-94.068,167.564,45.901,158.481
C03306=1026.881,-3.177,-94.053,167.561,45.903,158.481
C03307=1026.875,-3.427,-94.039,167.559,45.906,158.481
C03308=1026.869,-3.676,-94.024,167.556,45.908,158.481
C03309=1026.864,-3.926,-94.011,167.554,45.910,158.481
C03310=1026.856,-4.208,-93.994,167.551,45.913,158.481
C03311=1026.849,-4.491,-93.978,167.547,45.916,158.481
C03312=1026.842,-4.774,-93.963,167.545,45.918,158.482
C03313=1026.835,-5.056,-93.946,167.542,45.921,158.482
C03314=1026.829,-5.305,-93.933,167.539,45.924,158.482
C03315=1026.822,-5.555,-93.918,167.536,45.927,158.482
C03316=1026.816,-5.804,-93.905,167.534,45.929,158.482
C03317=1026.810,-6.054,-93.890,167.531,45.932,158.483
C03318=1026.804,-6.303,-93.876,167.529,45.935,158.483
C03319=1026.797,-6.553,-93.862,167.525,45.937,158.483
C03320=1026.792,-6.802,-93.848,167.523,45.940,158.483
C03321=1026.785,-7.052,-93.834,167.521,45.942,158.483
C03322=1026.779,-7.302,-93.820,167.517,45.945,158.483
C03323=1026.773,-7.550,-93.806,167.515,45.947,158.484
C03324=1026.767,-7.800,-93.792,167.513,45.949,158.484
C03325=1026.761,-8.050,-93.779,167.510,45.952,158.484
C03326=1026.754,-8.299,-93.764,167.507,45.955,158.484
C03327=1026.748,-8.549,-93.750,167.504,45.957,158.484
C03328=1026.742,-8.799,-93.736,167.502,45.960,158.485
C03329=1026.736,-9.048,-93.722,167.500,45.962,158.485
C03330=1026.730,-9.297,-93.708,167.496,45.965,158.485
C03331=1026.724,-9.547,-93.694,167.494,45.968,158.485
C03332=1026.718,-9.797,-93.681,167.491,45.970,158.485
C03333=1026.711,-10.046,-93.666,167.489,45.973,158.485
C03334=1026.705,-10.296,-93.653,167.486,45.975,158.485
C03335=1026.700,-10.545,-93.639,167.483,45.978,158.486
C03336=1026.692,-10.795,-93.624,167.481,45.980,158.486
C03337=1026.687,-11.044,-93.610,167.478,45.983,158.486
C03338=1026.680,-11.294,-93.597,167.475,45.985,158.486
C03339=1026.675,-11.544,-93.583,167.473,45.987,158.486
C03340=1026.668,-11.792,-93.569,167.470,45.990,158.487
C03341=1026.662,-12.043,-93.555,167.467,45.992,158.487
C03342=1026.657,-12.292,-93.541,167.465,45.995,158.487
C03343=1026.650,-12.541,-93.528,167.462,45.997,158.487
C03344=1026.644,-12.792,-93.513,167.460,46.000,158.487
C03345=1026.638,-13.040,-93.499,167.457,46.003,158.487
C03346=1026.632,-13.290,-93.486,167.454,46.005,158.487
C03347=1026.625,-13.540,-93.472,167.452,46.008,158.488
C03348=1026.620,-13.789,-93.458,167.449,46.010,158.488
C03349=1026.614,-14.039,-93.445,167.446,46.013,158.488
C03350=1026.608,-14.289,-93.431,167.443,46.015,158.488
C03351=1026.601,-14.538,-93.417,167.441,46.018,158.488
C03352=1026.596,-14.787,-93.403,167.437,46.020,158.488
C03353=1026.590,-15.036,-93.389,167.435,46.023,158.488
C03354=1026.583,-15.287,-93.375,167.433,46.025,158.489
C03355=1026.577,-15.536,-93.362,167.430,46.027,158.489
C03356=1026.572,-15.786,-93.348,167.427,46.030,158.489
C03357=1026.565,-16.036,-93.334,167.425,46.033,158.489
C03358=1026.559,-16.285,-93.321,167.422,46.035,158.489
C03359=1026.553,-16.534,-93.307,167.419,46.038,158.489
C03360=1026.546,-16.784,-93.294,167.416,46.040,158.490
C03361=1026.540,-17.034,-93.280,167.414,46.043,158.490
C03362=1026.534,-17.283,-93.267,167.411,46.045,158.490
C03363=1026.529,-17.532,-93.253,167.408,46.048,158.490
C03364=1026.522,-17.782,-93.240,167.406,46.051,158.490
C03365=1026.515,-18.032,-93.226,167.403,46.053,158.490
C03366=1026.509,-18.281,-93.213,167.400,46.056,158.491
C03367=1026.503,-18.531,-93.199,167.398,46.059,158.491
C03368=1026.497,-18.781,-93.186,167.394,46.061,158.491
C03369=1026.491,-19.030,-93.172,167.392,46.064,158.491
C03370=1026.485,-19.280,-93.160,167.390,46.066,158.491
C03371=1026.479,-19.530,-93.146,167.386,46.069,158.491
C03372=1026.473,-19.779,-93.132,167.384,46.072,158.492
C03373=1026.466,-20.028,-93.119,167.382,46.074,158.492
C03374=1026.460,-20.309,-93.104,167.378,46.077,158.492
C03375=1026.452,-20.590,-93.088,167.375,46.080,158.492
C03376=1026.446,-20.871,-93.073,167.372,46.083,158.492
C03377=1026.439,-21.151,-93.059,167.369,46.085,158.492
C03378=1026.432,-21.401,-93.045,167.366,46.088,158.493
C03379=1026.427,-21.650,-93.032,167.364,46.091,158.493
C03380=1026.420,-21.900,-93.018,167.361,46.093,158.493
C03381=1026.414,-22.150,-93.005,167.358,46.096,158.493
C03382=1026.408,-22.399,-92.992,167.355,46.098,158.493
C03383=1026.403,-22.649,-92.978,167.353,46.101,158.493
C03384=1026.396,-22.898,-92.965,167.350,46.103,158.493
C03385=1026.390,-23.148,-92.952,167.347,46.106,158.494
C03386=1026.384,-23.398,-92.939,167.345,46.109,158.494
C03387=1026.378,-23.648,-92.925,167.341,46.111,158.494
C03388=1026.372,-23.897,-92.912,167.339,46.114,158.494
C03389=1026.366,-24.146,-92.898,167.337,46.116,158.494
C03390=1026.360,-24.395,-92.885,167.333,46.119,158.494
C03391=1026.354,-24.645,-92.873,167.331,46.122,158.495
C03392=1026.348,-24.895,-92.859,167.329,46.124,158.495
C03393=1026.341,-25.145,-92.845,167.325,46.127,158.495
C03394=1026.335,-25.395,-92.832,167.323,46.129,158.495
C03395=1026.329,-25.644,-92.819,167.320,46.132,158.495
C03396=1026.324,-25.894,-92.805,167.317,46.134,158.495
C03397=1026.318,-26.143,-92.792,167.315,46.137,158.496
C03398=1026.312,-26.393,-92.780,167.312,46.139,158.496
C03399=1026.305,-26.642,-92.766,167.309,46.142,158.496
C03400=1026.299,-26.891,-92.753,167.306,46.144,158.496
C03401=1026.294,-27.141,-92.740,167.304,46.147,158.496
C03402=1026.288,-27.391,-92.727,167.301,46.150,158.496
C03403=1026.282,-27.640,-92.713,167.298,46.152,158.496
C03404=1026.275,-27.891,-92.700,167.295,46.155,158.497
C03405=1026.269,-28.140,-92.687,167.293,46.157,158.497
C03406=1026.263,-28.390,-92.675,167.290,46.159,158.497
C03407=1026.257,-28.639,-92.661,167.287,46.162,158.497
C03408=1026.251,-28.889,-92.649,167.285,46.165,158.497
C03409=1026.244,-29.138,-92.636,167.281,46.167,158.497
C03410=1026.238,-29.388,-92.623,167.279,46.170,158.498
C03411=1026.232,-29.637,-92.610,167.276,46.173,158.498
C03412=1026.226,-29.887,-92.598,167.273,46.176,158.498
C03413=1026.220,-30.136,-92.584,167.271,46.178,158.498
C03414=1026.214,-30.386,-92.572,167.267,46.181,158.498
C03415=1026.207,-30.635,-92.559,167.265,46.184,158.498
C03416=1026.202,-30.885,-92.546,167.263,46.186,158.499
C03417=1026.195,-31.134,-92.533,167.259,46.189,158.499
C03418=1026.189,-31.384,-92.520,167.257,46.192,158.499
C03419=1026.183,-31.634,-92.507,167.253,46.194,158.499
C03420=1026.177,-31.883,-92.494,167.251,46.197,158.499
C03421=1026.171,-32.133,-92.481,167.249,46.200,158.499
C03422=1026.165,-32.383,-92.469,167.245,46.202,158.499
C03423=1026.159,-32.633,-92.456,167.243,46.205,158.500
C03424=1026.153,-32.882,-92.443,167.240,46.207,158.500
C03425=1026.147,-33.132,-92.430,167.237,46.210,158.500
C03426=1026.140,-33.381,-92.417,167.234,46.213,158.500
C03427=1026.134,-33.630,-92.405,167.231,46.215,158.500
C03428=1026.128,-33.880,-92.392,167.229,46.218,158.500
C03429=1026.122,-34.130,-92.379,167.226,46.221,158.501
C03430=1026.116,-34.380,-92.367,167.223,46.223,158.501
C03431=1026.110,-34.629,-92.353,167.220,46.226,158.501
C03432=1026.104,-34.879,-92.341,167.218,46.228,158.501
C03433=1026.098,-35.129,-92.328,167.215,46.230,158.501
C03434=1026.092,-35.378,-92.315,167.212,46.233,158.501
C03435=1026.086,-35.628,-92.302,167.209,46.236,158.501
C03436=1026.080,-35.878,-92.290,167.206,46.239,158.502
C03437=1026.074,-36.127,-92.277,167.204,46.241,158.502
C03438=1026.067,-36.407,-92.263,167.200,46.244,158.502
C03439=1026.060,-36.687,-92.249,167.197,46.247,158.502
C03440=1026.054,-36.967,-92.235,167.195,46.249,158.502
C03441=1026.047,-37.247,-92.220,167.191,46.252,158.502
C03442=1026.042,-37.496,-92.208,167.188,46.255,158.502
C03443=1026.036,-37.746,-92.195,167.186,46.258,158.503
C03444=1026.029,-37.995,-92.182,167.182,46.261,158.503
C03445=1026.024,-38.245,-92.170,167.180,46.263,158.503
C03446=1026.017,-38.494,-92.158,167.178,46.265,158.503
C03447=1026.011,-38.744,-92.145,167.174,46.268,158.503
C03448=1026.005,-38.994,-92.132,167.172,46.271,158.503
C03449=1025.999,-39.243,-92.119,167.168,46.274,158.503
C03450=1025.993,-39.493,-92.107,167.166,46.276,158.504
C03451=1025.987,-39.742,-92.095,167.163,46.279,158.504
C03452=1025.981,-39.992,-92.083,167.160,46.281,158.504
C03453=1025.975,-40.242,-92.070,167.157,46.284,158.504
C03454=1025.968,-40.492,-92.058,167.155,46.287,158.504
C03455=1025.962,-40.741,-92.046,167.152,46.289,158.504
C03456=1025.957,-40.991,-92.033,167.149,46.292,158.505
C03457=1025.950,-41.241,-92.021,167.147,46.295,158.505
C03458=1025.945,-41.490,-92.009,167.143,46.298,158.505
C03459=1025.938,-41.739,-91.996,167.141,46.300,158.505
C03460=1025.932,-41.989,-91.984,167.138,46.303,158.505
C03461=1025.926,-42.239,-91.971,167.135,46.306,158.505
C03462=1025.919,-42.488,-91.959,167.132,46.308,158.505
C03463=1025.914,-42.738,-91.947,167.130,46.311,158.506
C03464=1025.908,-42.987,-91.934,167.126,46.314,158.506
C03465=1025.901,-43.237,-91.922,167.124,46.317,158.506
C03466=1025.895,-43.487,-91.910,167.120,46.319,158.506
C03467=1025.890,-43.737,-91.897,167.118,46.322,158.506
C03468=1025.883,-43.986,-91.886,167.115,46.325,158.506
C03469=1025.878,-44.236,-91.873,167.112,46.327,158.507
C03470=1025.872,-44.485,-91.861,167.109,46.330,158.507
C03471=1025.865,-44.735,-91.849,167.107,46.333,158.507
C03472=1025.860,-44.985,-91.837,167.103,46.335,158.507
C03473=1025.853,-45.234,-91.825,167.101,46.338,158.507
C03474=1025.847,-45.484,-91.813,167.098,46.341,158.507
C03475=1025.842,-45.734,-91.800,167.095,46.343,158.507
C03476=1025.836,-45.983,-91.788,167.092,46.346,158.508
C03477=1025.830,-46.233,-91.776,167.090,46.349,158.508
C03478=1025.824,-46.483,-91.763,167.086,46.351,158.508
C03479=1025.817,-46.732,-91.751,167.084,46.354,158.508
C03480=1025.812,-46.982,-91.739,167.082,46.357,158.508
C03481=1025.805,-47.231,-91.727,167.078,46.359,158.508
C03482=1025.799,-47.481,-91.715,167.076,46.362,158.509
C03483=1025.794,-47.731,-91.703,167.072,46.365,158.509
C03484=1025.788,-47.980,-91.691,167.070,46.367,158.509
C03485=1025.782,-48.230,-91.679,167.067,46.370,158.509
C03486=1025.776,-48.479,-91.667,167.064,46.373,158.509
C03487=1025.770,-48.729,-91.655,167.061,46.375,158.509
C03488=1025.764,-48.979,-91.642,167.059,46.378,158.509
C03489=1025.758,-49.228,-91.631,167.055,46.380,158.509
C03490=1025.752,-49.478,-91.619,167.053,46.383,158.510
C03491=1025.745,-49.728,-91.607,167.049,46.386,158.510
C03492=1025.740,-49.977,-91.594,167.047,46.388,158.510
C03493=1025.734,-50.227,-91.582,167.044,46.391,158.510
C03494=1025.728,-50.477,-91.571,167.041,46.394,158.510
C03495=1025.723,-50.726,-91.558,167.038,46.396,158.510
C03496=1025.716,-50.976,-91.546,167.036,46.399,158.510
C03497=1025.710,-51.226,-91.535,167.032,46.402,158.511
C03498=1025.704,-51.475,-91.523,167.030,46.405,158.511
C03499=1025.698,-51.725,-91.512,167.027,46.408,158.511
C03500=1025.691,-51.975,-91.500,167.023,46.411,158.511
C03501=1025.685,-52.224,-91.488,167.021,46.413,158.511
C03502=1025.678,-52.505,-91.476,167.018,46.417,158.512
C03503=1025.672,-52.785,-91.462,167.015,46.420,158.512
C03504=1025.665,-53.066,-91.449,167.011,46.423,158.512
C03505=1025.658,-53.346,-91.436,167.008,46.426,158.512
C03506=1025.652,-53.596,-91.425,167.005,46.429,158.512
C03507=1025.646,-53.845,-91.413,167.001,46.432,158.512
C03508=1025.640,-54.095,-91.401,166.999,46.435,158.513
C03509=1025.633,-54.345,-91.389,166.996,46.438,158.513
C03510=1025.627,-54.594,-91.378,166.994,46.441,158.513
C03511=1025.621,-54.844,-91.366,166.990,46.443,158.513
C03512=1025.616,-55.093,-91.354,166.988,46.446,158.513
C03513=1025.609,-55.343,-91.343,166.985,46.449,158.513
C03514=1025.603,-55.593,-91.331,166.981,46.452,158.513
C03515=1025.597,-55.842,-91.320,166.979,46.454,158.514
C03516=1025.590,-56.092,-91.309,166.976,46.458,158.514
C03517=1025.585,-56.342,-91.297,166.973,46.460,158.514
C03518=1025.579,-56.592,-91.286,166.970,46.463,158.514
C03519=1025.573,-56.841,-91.274,166.967,46.466,158.514
C03520=1025.566,-57.091,-91.263,166.964,46.468,158.514
C03521=1025.560,-57.340,-91.251,166.961,46.472,158.515
C03522=1025.555,-57.590,-91.239,166.959,46.474,158.515
C03523=1025.549,-57.839,-91.228,166.955,46.477,158.515
C03524=1025.542,-58.089,-91.216,166.952,46.480,158.515
C03525=1025.537,-58.339,-91.206,166.950,46.482,158.515
C03526=1025.530,-58.588,-91.194,166.947,46.486,158.515
C03527=1025.525,-58.838,-91.182,166.944,46.488,158.516
C03528=1025.519,-59.088,-91.171,166.941,46.491,158.516
C03529=1025.513,-59.337,-91.159,166.937,46.494,158.516
C03530=1025.506,-59.587,-91.148,166.935,46.496,158.516
C03531=1025.501,-59.837,-91.137,166.932,46.500,158.516
C03532=1025.494,-60.086,-91.125,166.930,46.502,158.516
C03533=1025.489,-60.336,-91.114,166.926,46.505,158.516
C03534=1025.483,-60.586,-91.103,166.924,46.507,158.517
C03535=1025.477,-60.835,-91.091,166.921,46.511,158.517
C03536=1025.470,-61.085,-91.080,166.917,46.514,158.517
C03537=1025.464,-61.335,-91.069,166.915,46.516,158.517
C03538=1025.458,-61.585,-91.057,166.911,46.519,158.517
C03539=1025.453,-61.834,-91.045,166.909,46.521,158.517
C03540=1025.447,-62.084,-91.034,166.906,46.525,158.517
C03541=1025.441,-62.334,-91.023,166.903,46.528,158.518
C03542=1025.435,-62.583,-91.012,166.900,46.530,158.518
C03543=1025.428,-62.833,-91.000,166.897,46.533,158.518
C03544=1025.423,-63.083,-90.990,166.895,46.536,158.518
C03545=1025.418,-63.332,-90.978,166.891,46.539,158.518
C03546=1025.411,-63.582,-90.966,166.888,46.541,158.518
C03547=1025.405,-63.831,-90.955,166.885,46.544,158.518
C03548=1025.399,-64.082,-90.944,166.882,46.547,158.519
C03549=1025.393,-64.331,-90.933,166.880,46.550,158.519
C03550=1025.387,-64.581,-90.922,166.876,46.552,158.519
C03551=1025.381,-64.831,-90.910,166.874,46.555,158.519
C03552=1025.376,-65.080,-90.899,166.871,46.558,158.519
C03553=1025.370,-65.329,-90.888,166.868,46.561,158.519
C03554=1025.364,-65.580,-90.877,166.865,46.563,158.519
///RCONF 1,0,0,1,0,0,0,0,0,0,0,0,0,0,0,0,0,0,0,0,0,0,0,0
C03555=1025.358,-65.829,-90.866,166.862,46.566,158.520
C03556=1025.352,-66.079,-90.855,166.860,46.569,158.520
C03557=1025.346,-66.328,-90.843,166.856,46.572,158.520
C03558=1025.341,-66.578,-90.831,166.853,46.574,158.520
C03559=1025.335,-66.828,-90.821,166.850,46.577,158.520
C03560=1025.328,-67.078,-90.809,166.847,46.580,158.520
C03561=1025.323,-67.327,-90.798,166.845,46.582,158.520
C03562=1025.317,-67.577,-90.788,166.841,46.585,158.520
C03563=1025.311,-67.826,-90.777,166.839,46.588,158.521
C03564=1025.305,-68.076,-90.765,166.836,46.591,158.521
C03565=1025.299,-68.326,-90.755,166.832,46.593,158.521
C03566=1025.293,-68.607,-90.741,166.829,46.596,158.521
C03567=1025.286,-68.889,-90.729,166.826,46.599,158.521
C03568=1025.280,-69.171,-90.717,166.822,46.602,158.521
C03569=1025.273,-69.451,-90.704,166.819,46.606,158.522
C03570=1025.267,-69.701,-90.693,166.817,46.608,158.522
C03571=1025.262,-69.951,-90.681,166.814,46.611,158.522
C03572=1025.256,-70.201,-90.671,166.810,46.614,158.522
C03573=1025.250,-70.450,-90.660,166.808,46.617,158.522
C03574=1025.244,-70.700,-90.648,166.805,46.620,158.522
C03575=1025.238,-70.950,-90.638,166.802,46.622,158.522
C03576=1025.232,-71.199,-90.627,166.799,46.625,158.522
C03577=1025.227,-71.449,-90.616,166.796,46.628,158.523
C03578=1025.221,-71.698,-90.605,166.793,46.631,158.523
C03579=1025.216,-71.949,-90.594,166.790,46.633,158.523
C03580=1025.210,-72.199,-90.583,166.787,46.636,158.523
C03581=1025.204,-72.448,-90.572,166.784,46.639,158.523
C03582=1025.198,-72.698,-90.561,166.782,46.641,158.523
C03583=1025.193,-72.947,-90.550,166.778,46.644,158.523
C03584=1025.187,-73.197,-90.539,166.776,46.647,158.524
